LIN {X 0,Y 407.799,Z 694.938,A -85,B 0,C 180,E1 -11054.266,E2 -11054.266} C_VEL
LIN {X 0,Y 407.045,Z 706.099,A -85,B 0,C 180,E1 -11055.216,E2 -11055.216} C_VEL
LIN {X 0,Y 406.273,Z 716.85,A -85,B 0,C 180,E1 -11056.367,E2 -11056.367} C_VEL
LIN {X 0,Y 406.01,Z 720.118,A -85,B 0,C 180,E1 -11056.773,E2 -11056.773} C_VEL
LIN {X 0,Y 404.973,Z 724.447,A -85,B 0,C 180,E1 -11057.328,E2 -11057.328} C_VEL
LIN {X 0,Y 401.518,Z 731.114,A -85,B 0,C 180,E1 -11058.251,E2 -11058.251} C_VEL
LIN {X 0,Y 398.157,Z 737.243,A -85,B 0,C 180,E1 -11059.262,E2 -11059.262} C_VEL
LIN {X 0,Y 397.276,Z 740.61,A -85,B 0,C 180,E1 -11059.945,E2 -11059.945} C_VEL
LIN {X 0,Y 396.697,Z 746.419,A -85,B 0,C 180,E1 -11061.338,E2 -11061.338} C_VEL
LIN {X 0,Y 396.363,Z 751.512,A -85,B 0,C 180,E1 -11062.869,E2 -11062.869} C_VEL
LIN {X 0,Y 396.152,Z 755.462,A -85,B 0,C 180,E1 -11064.4,E2 -11064.4} C_VEL
LIN {X 0,Y 395.896,Z 758.382,A -85,B 0,C 180,E1 -11065.927,E2 -11065.927} C_VEL
LIN {X 0,Y 395.868,Z 759.782,A -85,B 0,C 180,E1 -11066.946,E2 -11066.946} C_VEL
LIN {X 0,Y 395.86,Z 760.777,A -85,B 0,C 180,E1 -11067.964,E2 -11067.964} C_VEL
LIN {X 0,Y 395.779,Z 761.627,A -85,B 0,C 180,E1 -11069.999,E2 -11069.999} C_VEL
LIN {X 0,Y 395.797,Z 761.439,A -85,B 0,C 180,E1 -11071.017,E2 -11071.017} C_VEL
LIN {X 0,Y 395.86,Z 760.855,A -85,B 0,C 180,E1 -11072.034,E2 -11072.034} C_VEL
LIN {X 0,Y 395.886,Z 758.539,A -85,B 0,C 180,E1 -11074.071,E2 -11074.071} C_VEL
LIN {X 0,Y 396.142,Z 755.67,A -85,B 0,C 180,E1 -11075.599,E2 -11075.599} C_VEL
LIN {X 0,Y 396.361,Z 751.784,A -85,B 0,C 180,E1 -11077.129,E2 -11077.129} C_VEL
LIN {X 0,Y 396.687,Z 746.775,A -85,B 0,C 180,E1 -11078.66,E2 -11078.66} C_VEL
LIN {X 0,Y 397.268,Z 740.464,A -85,B 0,C 180,E1 -11080.189,E2 -11080.189} C_VEL
LIN {X 0,Y 397.969,Z 732.562,A -85,B 0,C 180,E1 -11081.716,E2 -11081.716} C_VEL
LIN {X 0,Y 398.706,Z 724.506,A -85,B 0,C 180,E1 -11082.987,E2 -11082.987} C_VEL
LIN {X 0,Y 399.608,Z 714.671,A -85,B 0,C 180,E1 -11084.253,E2 -11084.253} C_VEL
LIN {X 0,Y 400.355,Z 703.619,A -85,B 0,C 180,E1 -11085.396,E2 -11085.396} C_VEL
LIN {X 0,Y 401.175,Z 692.77,A -85,B 0,C 180,E1 -11086.277,E2 -11086.277} C_VEL
LIN {X 0,Y 401.93,Z 680.778,A -85,B 0,C 180,E1 -11087.03,E2 -11087.03} C_VEL
LIN {X 0,Y 402.452,Z 668.5,A -85,B 0,C 180,E1 -11087.596,E2 -11087.596} C_VEL
LIN {X 0,Y 402.857,Z 655.856,A -85,B 0,C 180,E1 -11087.972,E2 -11087.972} C_VEL
LIN {X 0,Y 403.735,Z 572.554,A -85,B 0,C 180,E1 -11089.479,E2 -11089.479} C_VEL
LIN {X 0,Y 399.424,Z 551.598,A -85,B 0,C 180,E1 -11090.112,E2 -11090.112} C_VEL
LIN {X 0,Y 399.354,Z 550.806,A -85,B 0,C 180,E1 -11090.204,E2 -11090.204} C_VEL
LIN {X 0,Y 399.28,Z 546.202,A -85,B 0,C 180,E1 -11091.342,E2 -11091.342} C_VEL
LIN {X 0,Y 397.408,Z 536.356,A -85,B 0,C 180,E1 -11093.999,E2 -11093.999} C_VEL
LIN {X 0,Y 397.147,Z 535.042,A -85,B 0,C 180,E1 -11094.433,E2 -11094.433} C_VEL
LIN {X 0,Y 397.161,Z 535.013,A -85,B 0,C 180,E1 -11097.775,E2 -11097.775} C_VEL
LIN {X 0,Y 397.077,Z 535.02,A -85,B 0,C 180,E1 -11100.881,E2 -11100.881} C_VEL
LIN {X 0,Y 397.124,Z 535.017,A -85,B 0,C 180,E1 -11104.492,E2 -11104.492} C_VEL
LIN {X 0,Y 397.104,Z 535.018,A -85,B 0,C 180,E1 -11108.273,E2 -11108.273} C_VEL
LIN {X 0,Y 397.103,Z 535.014,A -85,B 0,C 180,E1 -11110.905,E2 -11110.905} C_VEL
LIN {X 0,Y 397.099,Z 535.014,A -85,B 0,C 180,E1 -11113.647,E2 -11113.647} C_VEL
LIN {X 0,Y 397.1,Z 535.015,A -85,B 0,C 180,E1 -11116.52,E2 -11116.52} C_VEL
LIN {X 0,Y 397.116,Z 535.011,A -85,B 0,C 180,E1 -11119.55,E2 -11119.55} C_VEL
LIN {X 0,Y 397.094,Z 535.008,A -85,B 0,C 180,E1 -11122.789,E2 -11122.789} C_VEL
LIN {X 0,Y 397.113,Z 535.015,A -85,B 0,C 180,E1 -11126.281,E2 -11126.281} C_VEL
LIN {X 0,Y 397.108,Z 535.017,A -85,B 0,C 180,E1 -11130.132,E2 -11130.132} C_VEL
LIN {X 0,Y 397.188,Z 534.999,A -85,B 0,C 180,E1 -11132.609,E2 -11132.609} C_VEL
LIN {X 0,Y 397.126,Z 535.013,A -85,B 0,C 180,E1 -11135.981,E2 -11135.981} C_VEL
LIN {X 0,Y 397.137,Z 535.017,A -85,B 0,C 180,E1 -11139.702,E2 -11139.702} C_VEL
LIN {X 0,Y 397.174,Z 535.005,A -85,B 0,C 180,E1 -11142.844,E2 -11142.844} C_VEL
LIN {X 0,Y 397.221,Z 535.002,A -85,B 0,C 180,E1 -11146.702,E2 -11146.702} C_VEL
LIN {X 0,Y 397.211,Z 534.997,A -85,B 0,C 180,E1 -11149.809,E2 -11149.809} C_VEL
LIN {X 0,Y 397.356,Z 534.985,A -85,B 0,C 180,E1 -11152.888,E2 -11152.888} C_VEL
LIN {X 0,Y 397.249,Z 534.999,A -85,B 0,C 180,E1 -11154.925,E2 -11154.925} C_VEL
LIN {X 0,Y 397.444,Z 534.974,A -85,B 0,C 180,E1 -11157.973,E2 -11157.973} C_VEL
LIN {X 0,Y 397.575,Z 534.96,A -85,B 0,C 180,E1 -11160,E2 -11160} C_VEL
LIN {X 0,Y 397.375,Z 534.979,A -85,B 0,C 180,E1 -11163.041,E2 -11163.041} C_VEL
LIN {X 0,Y 397.377,Z 534.984,A -85,B 0,C 180,E1 -11166.091,E2 -11166.091} C_VEL
LIN {X 0,Y 397.369,Z 534.982,A -85,B 0,C 180,E1 -11168.134,E2 -11168.134} C_VEL
LIN {X 0,Y 397.221,Z 535.002,A -85,B 0,C 180,E1 -11172.258,E2 -11172.258} C_VEL
LIN {X 0,Y 397.172,Z 535.007,A -85,B 0,C 180,E1 -11175.392,E2 -11175.392} C_VEL
LIN {X 0,Y 397.164,Z 535.009,A -85,B 0,C 180,E1 -11178.573,E2 -11178.573} C_VEL
LIN {X 0,Y 397.103,Z 535.015,A -85,B 0,C 180,E1 -11181.818,E2 -11181.818} C_VEL
LIN {X 0,Y 397.146,Z 535.015,A -85,B 0,C 180,E1 -11185.513,E2 -11185.513} C_VEL
LIN {X 0,Y 397.115,Z 535.016,A -85,B 0,C 180,E1 -11188.544,E2 -11188.544} C_VEL
LIN {X 0,Y 397.074,Z 535.023,A -85,B 0,C 180,E1 -11192.072,E2 -11192.072} C_VEL
LIN {X 0,Y 397.114,Z 535.008,A -85,B 0,C 180,E1 -11195.504,E2 -11195.504} C_VEL
LIN {X 0,Y 397.128,Z 535.013,A -85,B 0,C 180,E1 -11198.863,E2 -11198.863} C_VEL
LIN {X 0,Y 397.063,Z 535.012,A -85,B 0,C 180,E1 -11202.268,E2 -11202.268} C_VEL
LIN {X 0,Y 397.112,Z 535.018,A -85,B 0,C 180,E1 -11205.065,E2 -11205.065} C_VEL
LIN {X 0,Y 397.152,Z 535.013,A -85,B 0,C 180,E1 -11208.008,E2 -11208.008} C_VEL
LIN {X 0,Y 397.106,Z 534.998,A -85,B 0,C 180,E1 -11211.727,E2 -11211.727} C_VEL
LIN {X 0,Y 397.123,Z 535.016,A -85,B 0,C 180,E1 -11215.508,E2 -11215.508} C_VEL
LIN {X 0,Y 397.075,Z 534.966,A -85,B 0,C 180,E1 -11219.119,E2 -11219.119} C_VEL
LIN {X 0,Y 397.218,Z 535.203,A -85,B 0,C 180,E1 -11221.661,E2 -11221.661} C_VEL
LIN {X 0,Y 399.624,Z 546.906,A -85,B 0,C 180,E1 -11224.478,E2 -11224.478} C_VEL
LIN {X 0,Y 400.536,Z 552.863,A -85,B 0,C 180,E1 -11225.842,E2 -11225.842} C_VEL
LIN {X 0,Y 399.226,Z 569.505,A -85,B 0,C 180,E1 -11229.386,E2 -11229.386} C_VEL
LIN {X 0,Y 399.065,Z 572.109,A -85,B 0,C 180,E1 -11229.883,E2 -11229.883} C_VEL
LIN {X 0,Y 403.53,Z 599.626,A -85,B 0,C 180,E1 -11230.651,E2 -11230.651} C_VEL
LIN {X 0,Y 402.595,Z 680.184,A -85,B 0,C 180,E1 -11232.115,E2 -11232.115} C_VEL
LIN {X 0,Y 401.967,Z 693.403,A -85,B 0,C 180,E1 -11232.546,E2 -11232.546} C_VEL
LIN {X 0,Y 401.348,Z 705.547,A -85,B 0,C 180,E1 -11233.142,E2 -11233.142} C_VEL
LIN {X 0,Y 400.486,Z 717.81,A -85,B 0,C 180,E1 -11233.956,E2 -11233.956} C_VEL
LIN {X 0,Y 399.547,Z 729.658,A -85,B 0,C 180,E1 -11234.99,E2 -11234.99} C_VEL
LIN {X 0,Y 398.735,Z 739.944,A -85,B 0,C 180,E1 -11236.119,E2 -11236.119} C_VEL
LIN {X 0,Y 398.055,Z 748.375,A -85,B 0,C 180,E1 -11237.251,E2 -11237.251} C_VEL
LIN {X 0,Y 397.306,Z 756.249,A -85,B 0,C 180,E1 -11238.522,E2 -11238.522} C_VEL
LIN {X 0,Y 396.689,Z 763.945,A -85,B 0,C 180,E1 -11240.054,E2 -11240.054} C_VEL
LIN {X 0,Y 396.226,Z 771.041,A -85,B 0,C 180,E1 -11241.843,E2 -11241.843} C_VEL
LIN {X 0,Y 395.936,Z 775.764,A -85,B 0,C 180,E1 -11243.376,E2 -11243.376} C_VEL
LIN {X 0,Y 395.851,Z 779.377,A -85,B 0,C 180,E1 -11244.908,E2 -11244.908} C_VEL
LIN {X 0,Y 395.778,Z 781.239,A -85,B 0,C 180,E1 -11245.928,E2 -11245.928} C_VEL
LIN {X 0,Y 395.763,Z 783.631,A -85,B 0,C 180,E1 -11247.966,E2 -11247.966} C_VEL
LIN {X 0,Y 395.778,Z 784.939,A -85,B 0,C 180,E1 -11250.001,E2 -11250.001} C_VEL
LIN {X 0,Y 395.773,Z 784.842,A -85,B 0,C 180,E1 -11251.018,E2 -11251.018} C_VEL
LIN {X 0,Y 395.761,Z 784.158,A -85,B 0,C 180,E1 -11252.036,E2 -11252.036} C_VEL
LIN {X 0,Y 395.729,Z 782.89,A -85,B 0,C 180,E1 -11253.055,E2 -11253.055} C_VEL
LIN {X 0,Y 395.852,Z 779.359,A -85,B 0,C 180,E1 -11255.094,E2 -11255.094} C_VEL
LIN {X 0,Y 395.921,Z 775.744,A -85,B 0,C 180,E1 -11256.626,E2 -11256.626} C_VEL
LIN {X 0,Y 396.228,Z 771.015,A -85,B 0,C 180,E1 -11258.159,E2 -11258.159} C_VEL
LIN {X 0,Y 396.691,Z 763.91,A -85,B 0,C 180,E1 -11259.948,E2 -11259.948} C_VEL
LIN {X 0,Y 397.308,Z 756.204,A -85,B 0,C 180,E1 -11261.479,E2 -11261.479} C_VEL
LIN {X 0,Y 398.22,Z 746.53,A -85,B 0,C 180,E1 -11263.005,E2 -11263.005} C_VEL
LIN {X 0,Y 398.974,Z 736.549,A -85,B 0,C 180,E1 -11264.278,E2 -11264.278} C_VEL
LIN {X 0,Y 399.861,Z 725.275,A -85,B 0,C 180,E1 -11265.418,E2 -11265.418} C_VEL
LIN {X 0,Y 400.714,Z 714.238,A -85,B 0,C 180,E1 -11266.298,E2 -11266.298} C_VEL
LIN {X 0,Y 401.554,Z 702.011,A -85,B 0,C 180,E1 -11267.048,E2 -11267.048} C_VEL
LIN {X 0,Y 402.233,Z 689.149,A -85,B 0,C 180,E1 -11267.608,E2 -11267.608} C_VEL
LIN {X 0,Y 402.671,Z 675.476,A -85,B 0,C 180,E1 -11267.982,E2 -11267.982} C_VEL
LIN {X 0,Y 403.517,Z 599.547,A -85,B 0,C 180,E1 -11269.344,E2 -11269.344} C_VEL
LIN {X 0,Y 399.119,Z 572.48,A -85,B 0,C 180,E1 -11270.083,E2 -11270.083} C_VEL
LIN {X 0,Y 399.14,Z 570.706,A -85,B 0,C 180,E1 -11270.351,E2 -11270.351} C_VEL
LIN {X 0,Y 400.427,Z 554.441,A -85,B 0,C 180,E1 -11273.809,E2 -11273.809} C_VEL
LIN {X 0,Y 400.428,Z 551.46,A -85,B 0,C 180,E1 -11274.462,E2 -11274.462} C_VEL
LIN {X 0,Y 398.096,Z 539.235,A -85,B 0,C 180,E1 -11277.324,E2 -11277.324} C_VEL
LIN {X 0,Y 397.202,Z 535.088,A -85,B 0,C 180,E1 -11278.391,E2 -11278.391} C_VEL
LIN {X 0,Y 397.082,Z 535.023,A -85,B 0,C 180,E1 -11282.072,E2 -11282.072} C_VEL
LIN {X 0,Y 397.123,Z 535.016,A -85,B 0,C 180,E1 -11285.504,E2 -11285.504} C_VEL
LIN {X 0,Y 397.133,Z 535.013,A -85,B 0,C 180,E1 -11288.862,E2 -11288.862} C_VEL
LIN {X 0,Y 397.073,Z 535.023,A -85,B 0,C 180,E1 -11292.267,E2 -11292.267} C_VEL
LIN {X 0,Y 397.091,Z 535.022,A -85,B 0,C 180,E1 -11295.069,E2 -11295.069} C_VEL
LIN {X 0,Y 397.07,Z 535.024,A -85,B 0,C 180,E1 -11298.021,E2 -11298.021} C_VEL
LIN {X 0,Y 397.135,Z 535.015,A -85,B 0,C 180,E1 -11301.139,E2 -11301.139} C_VEL
LIN {X 0,Y 397.124,Z 535.018,A -85,B 0,C 180,E1 -11304.497,E2 -11304.497} C_VEL
LIN {X 0,Y 397.082,Z 535.025,A -85,B 0,C 180,E1 -11307.929,E2 -11307.929} C_VEL
LIN {X 0,Y 397.153,Z 535.328,A -85,B 0,C 180,E1 -11308.441,E2 -11308.441} C_VEL
LIN {X 0,Y 400.671,Z 546.972,A -85,B 0,C 180,E1 -11310.865,E2 -11310.865} C_VEL
LIN {X 0,Y 402.695,Z 556.853,A -85,B 0,C 180,E1 -11312.734,E2 -11312.734} C_VEL
LIN {X 0,Y 402.289,Z 566.911,A -85,B 0,C 180,E1 -11314.381,E2 -11314.381} C_VEL
LIN {X 0,Y 400.826,Z 591.579,A -85,B 0,C 180,E1 -11318.395,E2 -11318.395} C_VEL
LIN {X 0,Y 399.629,Z 613.667,A -85,B 0,C 180,E1 -11321.956,E2 -11321.956} C_VEL
LIN {X 0,Y 398.858,Z 631.986,A -85,B 0,C 180,E1 -11324.878,E2 -11324.878} C_VEL
LIN {X 0,Y 400.775,Z 645.77,A -85,B 0,C 180,E1 -11325.351,E2 -11325.351} C_VEL
LIN {X 0,Y 400.953,Z 651.079,A -85,B 0,C 180,E1 -11325.497,E2 -11325.497} C_VEL
LIN {X 0,Y 399.755,Z 704.823,A -85,B 0,C 180,E1 -11326.788,E2 -11326.788} C_VEL
LIN {X 0,Y 399.417,Z 714.365,A -85,B 0,C 180,E1 -11327.165,E2 -11327.165} C_VEL
LIN {X 0,Y 398.946,Z 725.525,A -85,B 0,C 180,E1 -11327.796,E2 -11327.796} C_VEL
LIN {X 0,Y 398.427,Z 735.11,A -85,B 0,C 180,E1 -11328.554,E2 -11328.554} C_VEL
LIN {X 0,Y 397.928,Z 743.939,A -85,B 0,C 180,E1 -11329.442,E2 -11329.442} C_VEL
LIN {X 0,Y 397.309,Z 752.78,A -85,B 0,C 180,E1 -11330.583,E2 -11330.583} C_VEL
LIN {X 0,Y 396.852,Z 759.018,A -85,B 0,C 180,E1 -11331.599,E2 -11331.599} C_VEL
LIN {X 0,Y 396.59,Z 764.139,A -85,B 0,C 180,E1 -11332.618,E2 -11332.618} C_VEL
LIN {X 0,Y 396.36,Z 769.29,A -85,B 0,C 180,E1 -11333.893,E2 -11333.893} C_VEL
LIN {X 0,Y 395.965,Z 773.837,A -85,B 0,C 180,E1 -11335.419,E2 -11335.419} C_VEL
LIN {X 0,Y 395.831,Z 776.856,A -85,B 0,C 180,E1 -11336.947,E2 -11336.947} C_VEL
LIN {X 0,Y 395.795,Z 778.116,A -85,B 0,C 180,E1 -11337.965,E2 -11337.965} C_VEL
LIN {X 0,Y 395.76,Z 778.793,A -85,B 0,C 180,E1 -11338.983,E2 -11338.983} C_VEL
LIN {X 0,Y 395.76,Z 778.896,A -85,B 0,C 180,E1 -11340,E2 -11340} C_VEL
LIN {X 0,Y 395.76,Z 778.422,A -85,B 0,C 180,E1 -11341.018,E2 -11341.018} C_VEL
LIN {X 0,Y 395.772,Z 777.361,A -85,B 0,C 180,E1 -11342.035,E2 -11342.035} C_VEL
LIN {X 0,Y 395.824,Z 774.538,A -85,B 0,C 180,E1 -11343.563,E2 -11343.563} C_VEL
LIN {X 0,Y 395.99,Z 770.335,A -85,B 0,C 180,E1 -11345.091,E2 -11345.091} C_VEL
LIN {X 0,Y 396.141,Z 764.731,A -85,B 0,C 180,E1 -11346.53,E2 -11346.53} C_VEL
LIN {X 0,Y 396.444,Z 759.18,A -85,B 0,C 180,E1 -11347.641,E2 -11347.641} C_VEL
LIN {X 0,Y 396.687,Z 752.914,A -85,B 0,C 180,E1 -11348.661,E2 -11348.661} C_VEL
LIN {X 0,Y 397.099,Z 744.072,A -85,B 0,C 180,E1 -11349.808,E2 -11349.808} C_VEL
LIN {X 0,Y 397.525,Z 735.203,A -85,B 0,C 180,E1 -11350.698,E2 -11350.698} C_VEL
LIN {X 0,Y 397.944,Z 725.554,A -85,B 0,C 180,E1 -11351.46,E2 -11351.46} C_VEL
LIN {X 0,Y 398.193,Z 715.643,A -85,B 0,C 180,E1 -11352.034,E2 -11352.034} C_VEL
LIN {X 0,Y 398.502,Z 705.429,A -85,B 0,C 180,E1 -11352.444,E2 -11352.444} C_VEL
LIN {X 0,Y 398.767,Z 689.785,A -85,B 0,C 180,E1 -11352.824,E2 -11352.824} C_VEL
LIN {X 0,Y 399.26,Z 646.715,A -85,B 0,C 180,E1 -11353.772,E2 -11353.772} C_VEL
LIN {X 0,Y 397.778,Z 631.757,A -85,B 0,C 180,E1 -11354.162,E2 -11354.162} C_VEL
LIN {X 0,Y 398.287,Z 617.682,A -85,B 0,C 180,E1 -11356.399,E2 -11356.399} C_VEL
LIN {X 0,Y 399.179,Z 596.662,A -85,B 0,C 180,E1 -11359.811,E2 -11359.811} C_VEL
LIN {X 0,Y 400.154,Z 575.39,A -85,B 0,C 180,E1 -11363.277,E2 -11363.277} C_VEL
LIN {X 0,Y 401.199,Z 556.319,A -85,B 0,C 180,E1 -11366.384,E2 -11366.384} C_VEL
LIN {X 0,Y 400.728,Z 551.948,A -85,B 0,C 180,E1 -11367.129,E2 -11367.129} C_VEL
LIN {X 0,Y 397.187,Z 535.186,A -85,B 0,C 180,E1 -11370.129,E2 -11370.129} C_VEL
LIN {X 0,Y 397.123,Z 535.018,A -85,B 0,C 180,E1 -11373.718,E2 -11373.718} C_VEL
LIN {X 0,Y 397.102,Z 535.018,A -85,B 0,C 180,E1 -11377.209,E2 -11377.209} C_VEL
LIN {X 0,Y 397.106,Z 535.008,A -85,B 0,C 180,E1 -11380.445,E2 -11380.445} C_VEL
LIN {X 0,Y 397.105,Z 534.994,A -85,B 0,C 180,E1 -11383.648,E2 -11383.648} C_VEL
LIN {X 0,Y 397.111,Z 535.02,A -85,B 0,C 180,E1 -11386.52,E2 -11386.52} C_VEL
LIN {X 0,Y 397.117,Z 534.998,A -85,B 0,C 180,E1 -11390.422,E2 -11390.422} C_VEL
LIN {X 0,Y 397.112,Z 535.02,A -85,B 0,C 180,E1 -11394.265,E2 -11394.265} C_VEL
LIN {X 0,Y 397.119,Z 535.017,A -85,B 0,C 180,E1 -11396.727,E2 -11396.727} C_VEL
LIN {X 0,Y 397.129,Z 535.019,A -85,B 0,C 180,E1 -11400.295,E2 -11400.295} C_VEL
LIN {X 0,Y 397.199,Z 535.011,A -85,B 0,C 180,E1 -11402.609,E2 -11402.609} C_VEL
LIN {X 0,Y 397.183,Z 535.091,A -85,B 0,C 180,E1 -11405.706,E2 -11405.706} C_VEL
LIN {X 0,Y 399.242,Z 545.825,A -85,B 0,C 180,E1 -11408.659,E2 -11408.659} C_VEL
LIN {X 0,Y 399.384,Z 550.325,A -85,B 0,C 180,E1 -11409.797,E2 -11409.797} C_VEL
LIN {X 0,Y 399.383,Z 551.427,A -85,B 0,C 180,E1 -11409.978,E2 -11409.978} C_VEL
LIN {X 0,Y 403.8,Z 572.909,A -85,B 0,C 180,E1 -11410.629,E2 -11410.629} C_VEL
LIN {X 0,Y 402.826,Z 655.828,A -85,B 0,C 180,E1 -11412.123,E2 -11412.123} C_VEL
LIN {X 0,Y 402.425,Z 668.491,A -85,B 0,C 180,E1 -11412.499,E2 -11412.499} C_VEL
LIN {X 0,Y 401.831,Z 681.338,A -85,B 0,C 180,E1 -11413.095,E2 -11413.095} C_VEL
LIN {X 0,Y 401.117,Z 693.197,A -85,B 0,C 180,E1 -11413.85,E2 -11413.85} C_VEL
LIN {X 0,Y 400.352,Z 703.959,A -85,B 0,C 180,E1 -11414.732,E2 -11414.732} C_VEL
LIN {X 0,Y 399.589,Z 714.927,A -85,B 0,C 180,E1 -11415.874,E2 -11415.874} C_VEL
LIN {X 0,Y 398.584,Z 725.605,A -85,B 0,C 180,E1 -11417.266,E2 -11417.266} C_VEL
LIN {X 0,Y 397.941,Z 733.475,A -85,B 0,C 180,E1 -11418.539,E2 -11418.539} C_VEL
LIN {X 0,Y 397.276,Z 740.61,A -85,B 0,C 180,E1 -11419.945,E2 -11419.945} C_VEL
LIN {X 0,Y 396.419,Z 743.788,A -85,B 0,C 180,E1 -11420.653,E2 -11420.653} C_VEL
LIN {X 0,Y 393.189,Z 748.517,A -85,B 0,C 180,E1 -11421.826,E2 -11421.826} C_VEL
LIN {X 0,Y 389.965,Z 752.575,A -85,B 0,C 180,E1 -11423.067,E2 -11423.067} C_VEL
LIN {X 0,Y 389.14,Z 754.668,A -85,B 0,C 180,E1 -11423.873,E2 -11423.873} C_VEL
LIN {X 0,Y 388.822,Z 758.588,A -85,B 0,C 180,E1 -11425.853,E2 -11425.853} C_VEL
LIN {X 0,Y 388.772,Z 759.987,A -85,B 0,C 180,E1 -11426.89,E2 -11426.89} C_VEL
LIN {X 0,Y 388.763,Z 760.982,A -85,B 0,C 180,E1 -11427.927,E2 -11427.927} C_VEL
LIN {X 0,Y 388.708,Z 761.831,A -85,B 0,C 180,E1 -11429.999,E2 -11429.999} C_VEL
LIN {X 0,Y 388.728,Z 761.643,A -85,B 0,C 180,E1 -11431.035,E2 -11431.035} C_VEL
LIN {X 0,Y 388.762,Z 761.06,A -85,B 0,C 180,E1 -11432.071,E2 -11432.071} C_VEL
LIN {X 0,Y 388.812,Z 758.743,A -85,B 0,C 180,E1 -11434.145,E2 -11434.145} C_VEL
LIN {X 0,Y 389.075,Z 755.874,A -85,B 0,C 180,E1 -11435.701,E2 -11435.701} C_VEL
LIN {X 0,Y 389.312,Z 751.987,A -85,B 0,C 180,E1 -11437.259,E2 -11437.259} C_VEL
LIN {X 0,Y 389.672,Z 746.978,A -85,B 0,C 180,E1 -11438.817,E2 -11438.817} C_VEL
LIN {X 0,Y 390.281,Z 740.667,A -85,B 0,C 180,E1 -11440.373,E2 -11440.373} C_VEL
LIN {X 0,Y 391.009,Z 732.764,A -85,B 0,C 180,E1 -11441.928,E2 -11441.928} C_VEL
LIN {X 0,Y 391.804,Z 724.707,A -85,B 0,C 180,E1 -11443.22,E2 -11443.22} C_VEL
LIN {X 0,Y 392.723,Z 714.872,A -85,B 0,C 180,E1 -11444.508,E2 -11444.508} C_VEL
LIN {X 0,Y 393.51,Z 703.818,A -85,B 0,C 180,E1 -11445.671,E2 -11445.671} C_VEL
LIN {X 0,Y 394.387,Z 692.968,A -85,B 0,C 180,E1 -11446.565,E2 -11446.565} C_VEL
LIN {X 0,Y 395.159,Z 680.975,A -85,B 0,C 180,E1 -11447.331,E2 -11447.331} C_VEL
LIN {X 0,Y 395.712,Z 668.692,A -85,B 0,C 180,E1 -11447.906,E2 -11447.906} C_VEL
LIN {X 0,Y 396.129,Z 656.038,A -85,B 0,C 180,E1 -11448.288,E2 -11448.288} C_VEL
LIN {X 0,Y 397.126,Z 573.966,A -85,B 0,C 180,E1 -11449.793,E2 -11449.793} C_VEL
LIN {X 0,Y 392.54,Z 551.801,A -85,B 0,C 180,E1 -11450.48,E2 -11450.48} C_VEL
LIN {X 0,Y 392.484,Z 551.002,A -85,B 0,C 180,E1 -11450.573,E2 -11450.573} C_VEL
LIN {X 0,Y 392.23,Z 546.783,A -85,B 0,C 180,E1 -11451.647,E2 -11451.647} C_VEL
LIN {X 0,Y 390.217,Z 536.551,A -85,B 0,C 180,E1 -11454.47,E2 -11454.47} C_VEL
LIN {X 0,Y 390.124,Z 535.905,A -85,B 0,C 180,E1 -11454.76,E2 -11454.76} C_VEL
LIN {X 0,Y 390.095,Z 535.892,A -85,B 0,C 180,E1 -11458.019,E2 -11458.019} C_VEL
LIN {X 0,Y 390.022,Z 535.905,A -85,B 0,C 180,E1 -11461.503,E2 -11461.503} C_VEL
LIN {X 0,Y 390.066,Z 535.898,A -85,B 0,C 180,E1 -11464.024,E2 -11464.024} C_VEL
LIN {X 0,Y 390.043,Z 535.903,A -85,B 0,C 180,E1 -11467.55,E2 -11467.55} C_VEL
LIN {X 0,Y 390.068,Z 535.89,A -85,B 0,C 180,E1 -11470.823,E2 -11470.823} C_VEL
LIN {X 0,Y 390.053,Z 535.889,A -85,B 0,C 180,E1 -11473.885,E2 -11473.885} C_VEL
LIN {X 0,Y 390.076,Z 535.898,A -85,B 0,C 180,E1 -11477.619,E2 -11477.619} C_VEL
LIN {X 0,Y 390.09,Z 535.878,A -85,B 0,C 180,E1 -11480.907,E2 -11480.907} C_VEL
LIN {X 0,Y 390.081,Z 535.892,A -85,B 0,C 180,E1 -11484.792,E2 -11484.792} C_VEL
LIN {X 0,Y 390.021,Z 535.897,A -85,B 0,C 180,E1 -11488.495,E2 -11488.495} C_VEL
LIN {X 0,Y 390.11,Z 535.882,A -85,B 0,C 180,E1 -11492.069,E2 -11492.069} C_VEL
LIN {X 0,Y 390.074,Z 535.897,A -85,B 0,C 180,E1 -11495.519,E2 -11495.519} C_VEL
LIN {X 0,Y 390.054,Z 535.89,A -85,B 0,C 180,E1 -11498.878,E2 -11498.878} C_VEL
LIN {X 0,Y 390.121,Z 535.883,A -85,B 0,C 180,E1 -11502.166,E2 -11502.166} C_VEL
LIN {X 0,Y 390.136,Z 535.883,A -85,B 0,C 180,E1 -11505.392,E2 -11505.392} C_VEL
LIN {X 0,Y 390.141,Z 535.881,A -85,B 0,C 180,E1 -11508.571,E2 -11508.571} C_VEL
LIN {X 0,Y 390.336,Z 535.861,A -85,B 0,C 180,E1 -11511.993,E2 -11511.993} C_VEL
LIN {X 0,Y 390.221,Z 535.874,A -85,B 0,C 180,E1 -11514.833,E2 -11514.833} C_VEL
LIN {X 0,Y 390.413,Z 535.85,A -85,B 0,C 180,E1 -11517.937,E2 -11517.937} C_VEL
LIN {X 0,Y 390.544,Z 535.836,A -85,B 0,C 180,E1 -11520,E2 -11520} C_VEL
LIN {X 0,Y 390.309,Z 535.86,A -85,B 0,C 180,E1 -11523.097,E2 -11523.097} C_VEL
LIN {X 0,Y 390.33,Z 535.861,A -85,B 0,C 180,E1 -11526.202,E2 -11526.202} C_VEL
LIN {X 0,Y 390.307,Z 535.861,A -85,B 0,C 180,E1 -11528.282,E2 -11528.282} C_VEL
LIN {X 0,Y 390.17,Z 535.88,A -85,B 0,C 180,E1 -11532.483,E2 -11532.483} C_VEL
LIN {X 0,Y 390.132,Z 535.881,A -85,B 0,C 180,E1 -11535.677,E2 -11535.677} C_VEL
LIN {X 0,Y 390.109,Z 535.889,A -85,B 0,C 180,E1 -11538.922,E2 -11538.922} C_VEL
LIN {X 0,Y 390.041,Z 535.894,A -85,B 0,C 180,E1 -11542.234,E2 -11542.234} C_VEL
LIN {X 0,Y 390.112,Z 535.887,A -85,B 0,C 180,E1 -11545.744,E2 -11545.744} C_VEL
LIN {X 0,Y 390.052,Z 535.898,A -85,B 0,C 180,E1 -11549.11,E2 -11549.11} C_VEL
LIN {X 0,Y 390.037,Z 535.898,A -85,B 0,C 180,E1 -11552.722,E2 -11552.722} C_VEL
LIN {X 0,Y 390.051,Z 535.883,A -85,B 0,C 180,E1 -11555.826,E2 -11555.826} C_VEL
LIN {X 0,Y 390.066,Z 535.895,A -85,B 0,C 180,E1 -11559.22,E2 -11559.22} C_VEL
LIN {X 0,Y 390.037,Z 535.887,A -85,B 0,C 180,E1 -11562.375,E2 -11562.375} C_VEL
LIN {X 0,Y 390.097,Z 535.887,A -85,B 0,C 180,E1 -11566.108,E2 -11566.108} C_VEL
LIN {X 0,Y 390.079,Z 535.895,A -85,B 0,C 180,E1 -11569.175,E2 -11569.175} C_VEL
LIN {X 0,Y 390.044,Z 535.876,A -85,B 0,C 180,E1 -11572.449,E2 -11572.449} C_VEL
LIN {X 0,Y 390.065,Z 535.888,A -85,B 0,C 180,E1 -11575.976,E2 -11575.976} C_VEL
LIN {X 0,Y 390.035,Z 535.847,A -85,B 0,C 180,E1 -11579.701,E2 -11579.701} C_VEL
LIN {X 0,Y 390.136,Z 536.007,A -85,B 0,C 180,E1 -11581.309,E2 -11581.309} C_VEL
LIN {X 0,Y 392.112,Z 545.401,A -85,B 0,C 180,E1 -11583.66,E2 -11583.66} C_VEL
LIN {X 0,Y 393.588,Z 553.612,A -85,B 0,C 180,E1 -11585.598,E2 -11585.598} C_VEL
LIN {X 0,Y 392.572,Z 566.29,A -85,B 0,C 180,E1 -11588.356,E2 -11588.356} C_VEL
LIN {X 0,Y 392.171,Z 571.907,A -85,B 0,C 180,E1 -11589.513,E2 -11589.513} C_VEL
LIN {X 0,Y 396.631,Z 598.893,A -85,B 0,C 180,E1 -11590.29,E2 -11590.29} C_VEL
LIN {X 0,Y 396.898,Z 604.479,A -85,B 0,C 180,E1 -11590.409,E2 -11590.409} C_VEL
LIN {X 0,Y 395.847,Z 679.991,A -85,B 0,C 180,E1 -11591.799,E2 -11591.799} C_VEL
LIN {X 0,Y 395.19,Z 693.206,A -85,B 0,C 180,E1 -11592.237,E2 -11592.237} C_VEL
LIN {X 0,Y 394.542,Z 705.348,A -85,B 0,C 180,E1 -11592.842,E2 -11592.842} C_VEL
LIN {X 0,Y 393.66,Z 717.61,A -85,B 0,C 180,E1 -11593.67,E2 -11593.67} C_VEL
LIN {X 0,Y 392.709,Z 729.2,A -85,B 0,C 180,E1 -11594.696,E2 -11594.696} C_VEL
LIN {X 0,Y 391.826,Z 739.797,A -85,B 0,C 180,E1 -11595.876,E2 -11595.876} C_VEL
LIN {X 0,Y 391.118,Z 748.172,A -85,B 0,C 180,E1 -11597.021,E2 -11597.021} C_VEL
LIN {X 0,Y 390.316,Z 756.045,A -85,B 0,C 180,E1 -11598.314,E2 -11598.314} C_VEL
LIN {X 0,Y 389.672,Z 763.741,A -85,B 0,C 180,E1 -11599.873,E2 -11599.873} C_VEL
LIN {X 0,Y 389.158,Z 770.836,A -85,B 0,C 180,E1 -11601.694,E2 -11601.694} C_VEL
LIN {X 0,Y 388.852,Z 775.558,A -85,B 0,C 180,E1 -11603.254,E2 -11603.254} C_VEL
LIN {X 0,Y 388.746,Z 779.172,A -85,B 0,C 180,E1 -11604.815,E2 -11604.815} C_VEL
LIN {X 0,Y 388.703,Z 781.035,A -85,B 0,C 180,E1 -11605.854,E2 -11605.854} C_VEL
LIN {X 0,Y 388.661,Z 783.428,A -85,B 0,C 180,E1 -11607.928,E2 -11607.928} C_VEL
LIN {X 0,Y 388.703,Z 784.331,A -85,B 0,C 180,E1 -11608.965,E2 -11608.965} C_VEL
LIN {X 0,Y 388.707,Z 784.857,A -85,B 0,C 180,E1 -11610.001,E2 -11610.001} C_VEL
LIN {X 0,Y 388.672,Z 784.808,A -85,B 0,C 180,E1 -11611.037,E2 -11611.037} C_VEL
LIN {X 0,Y 388.658,Z 784.172,A -85,B 0,C 180,E1 -11612.073,E2 -11612.073} C_VEL
LIN {X 0,Y 388.636,Z 782.944,A -85,B 0,C 180,E1 -11613.111,E2 -11613.111} C_VEL
LIN {X 0,Y 388.733,Z 777.962,A -85,B 0,C 180,E1 -11615.762,E2 -11615.762} C_VEL
LIN {X 0,Y 388.942,Z 774.103,A -85,B 0,C 180,E1 -11617.267,E2 -11617.267} C_VEL
LIN {X 0,Y 389.357,Z 767.984,A -85,B 0,C 180,E1 -11619.088,E2 -11619.088} C_VEL
LIN {X 0,Y 389.881,Z 761.302,A -85,B 0,C 180,E1 -11620.648,E2 -11620.648} C_VEL
LIN {X 0,Y 390.633,Z 753.015,A -85,B 0,C 180,E1 -11622.205,E2 -11622.205} C_VEL
LIN {X 0,Y 391.403,Z 744.52,A -85,B 0,C 180,E1 -11623.5,E2 -11623.5} C_VEL
LIN {X 0,Y 392.242,Z 734.022,A -85,B 0,C 180,E1 -11624.794,E2 -11624.794} C_VEL
LIN {X 0,Y 393.136,Z 723.638,A -85,B 0,C 180,E1 -11625.821,E2 -11625.821} C_VEL
LIN {X 0,Y 394.061,Z 712.261,A -85,B 0,C 180,E1 -11626.714,E2 -11626.714} C_VEL
LIN {X 0,Y 394.828,Z 700.579,A -85,B 0,C 180,E1 -11627.414,E2 -11627.414} C_VEL
LIN {X 0,Y 395.562,Z 687.102,A -85,B 0,C 180,E1 -11627.982,E2 -11627.982} C_VEL
LIN {X 0,Y 395.981,Z 673.712,A -85,B 0,C 180,E1 -11628.33,E2 -11628.33} C_VEL
LIN {X 0,Y 396.796,Z 600.305,A -85,B 0,C 180,E1 -11629.666,E2 -11629.666} C_VEL
LIN {X 0,Y 392.212,Z 571.997,A -85,B 0,C 180,E1 -11630.469,E2 -11630.469} C_VEL
LIN {X 0,Y 392.46,Z 567.476,A -85,B 0,C 180,E1 -11631.378,E2 -11631.378} C_VEL
LIN {X 0,Y 393.635,Z 554.251,A -85,B 0,C 180,E1 -11634.246,E2 -11634.246} C_VEL
LIN {X 0,Y 392.105,Z 545.375,A -85,B 0,C 180,E1 -11636.338,E2 -11636.338} C_VEL
LIN {X 0,Y 390.189,Z 536.144,A -85,B 0,C 180,E1 -11638.621,E2 -11638.621} C_VEL
LIN {X 0,Y 390.092,Z 535.868,A -85,B 0,C 180,E1 -11639.108,E2 -11639.108} C_VEL
LIN {X 0,Y 390.047,Z 535.901,A -85,B 0,C 180,E1 -11642.722,E2 -11642.722} C_VEL
LIN {X 0,Y 390.06,Z 535.897,A -85,B 0,C 180,E1 -11645.826,E2 -11645.826} C_VEL
LIN {X 0,Y 390.073,Z 535.893,A -85,B 0,C 180,E1 -11649.219,E2 -11649.219} C_VEL
LIN {X 0,Y 390.046,Z 535.898,A -85,B 0,C 180,E1 -11652.375,E2 -11652.375} C_VEL
LIN {X 0,Y 390.048,Z 535.9,A -85,B 0,C 180,E1 -11655.355,E2 -11655.355} C_VEL
LIN {X 0,Y 390.035,Z 535.901,A -85,B 0,C 180,E1 -11658.187,E2 -11658.187} C_VEL
LIN {X 0,Y 390.095,Z 535.892,A -85,B 0,C 180,E1 -11660.908,E2 -11660.908} C_VEL
LIN {X 0,Y 390.09,Z 535.894,A -85,B 0,C 180,E1 -11664.794,E2 -11664.794} C_VEL
LIN {X 0,Y 390.071,Z 536.13,A -85,B 0,C 180,E1 -11667.712,E2 -11667.712} C_VEL
LIN {X 0,Y 393.337,Z 546.37,A -85,B 0,C 180,E1 -11669.98,E2 -11669.98} C_VEL
LIN {X 0,Y 395.349,Z 554.413,A -85,B 0,C 180,E1 -11671.607,E2 -11671.607} C_VEL
LIN {X 0,Y 396.227,Z 560.862,A -85,B 0,C 180,E1 -11672.804,E2 -11672.804} C_VEL
LIN {X 0,Y 394.864,Z 580.85,A -85,B 0,C 180,E1 -11676.114,E2 -11676.114} C_VEL
LIN {X 0,Y 393.769,Z 598.994,A -85,B 0,C 180,E1 -11679.086,E2 -11679.086} C_VEL
LIN {X 0,Y 392.542,Z 621.651,A -85,B 0,C 180,E1 -11682.818,E2 -11682.818} C_VEL
LIN {X 0,Y 392.053,Z 631.777,A -85,B 0,C 180,E1 -11684.46,E2 -11684.46} C_VEL
LIN {X 0,Y 393.839,Z 644.005,A -85,B 0,C 180,E1 -11684.923,E2 -11684.923} C_VEL
LIN {X 0,Y 394.362,Z 650.095,A -85,B 0,C 180,E1 -11685.113,E2 -11685.113} C_VEL
LIN {X 0,Y 393.043,Z 704.735,A -85,B 0,C 180,E1 -11686.46,E2 -11686.46} C_VEL
LIN {X 0,Y 392.628,Z 714.914,A -85,B 0,C 180,E1 -11686.873,E2 -11686.873} C_VEL
LIN {X 0,Y 392.203,Z 724.906,A -85,B 0,C 180,E1 -11687.451,E2 -11687.451} C_VEL
LIN {X 0,Y 391.621,Z 734.613,A -85,B 0,C 180,E1 -11688.221,E2 -11688.221} C_VEL
LIN {X 0,Y 391.171,Z 742.32,A -85,B 0,C 180,E1 -11688.995,E2 -11688.995} C_VEL
LIN {X 0,Y 390.591,Z 749.696,A -85,B 0,C 180,E1 -11689.896,E2 -11689.896} C_VEL
LIN {X 0,Y 389.968,Z 758.074,A -85,B 0,C 180,E1 -11691.188,E2 -11691.188} C_VEL
LIN {X 0,Y 389.65,Z 763.372,A -85,B 0,C 180,E1 -11692.225,E2 -11692.225} C_VEL
LIN {X 0,Y 389.327,Z 768.622,A -85,B 0,C 180,E1 -11693.504,E2 -11693.504} C_VEL
LIN {X 0,Y 389.032,Z 772.798,A -85,B 0,C 180,E1 -11694.818,E2 -11694.818} C_VEL
LIN {X 0,Y 388.817,Z 775.246,A -85,B 0,C 180,E1 -11695.854,E2 -11695.854} C_VEL
LIN {X 0,Y 388.737,Z 777.05,A -85,B 0,C 180,E1 -11696.891,E2 -11696.891} C_VEL
LIN {X 0,Y 388.698,Z 778.254,A -85,B 0,C 180,E1 -11697.928,E2 -11697.928} C_VEL
LIN {X 0,Y 388.66,Z 778.878,A -85,B 0,C 180,E1 -11698.964,E2 -11698.964} C_VEL
LIN {X 0,Y 388.672,Z 778.928,A -85,B 0,C 180,E1 -11700,E2 -11700} C_VEL
LIN {X 0,Y 388.66,Z 778.401,A -85,B 0,C 180,E1 -11701.036,E2 -11701.036} C_VEL
LIN {X 0,Y 388.671,Z 777.293,A -85,B 0,C 180,E1 -11702.073,E2 -11702.073} C_VEL
LIN {X 0,Y 388.738,Z 774.403,A -85,B 0,C 180,E1 -11703.628,E2 -11703.628} C_VEL
LIN {X 0,Y 388.868,Z 771.681,A -85,B 0,C 180,E1 -11704.665,E2 -11704.665} C_VEL
LIN {X 0,Y 388.942,Z 768.227,A -85,B 0,C 180,E1 -11705.704,E2 -11705.704} C_VEL
LIN {X 0,Y 389.197,Z 762.779,A -85,B 0,C 180,E1 -11707.001,E2 -11707.001} C_VEL
LIN {X 0,Y 389.481,Z 755.731,A -85,B 0,C 180,E1 -11708.3,E2 -11708.3} C_VEL
LIN {X 0,Y 389.824,Z 748.577,A -85,B 0,C 180,E1 -11709.338,E2 -11709.338} C_VEL
LIN {X 0,Y 390.285,Z 739.727,A -85,B 0,C 180,E1 -11710.374,E2 -11710.374} C_VEL
LIN {X 0,Y 390.738,Z 729.517,A -85,B 0,C 180,E1 -11711.28,E2 -11711.28} C_VEL
LIN {X 0,Y 391.083,Z 719.927,A -85,B 0,C 180,E1 -11711.927,E2 -11711.927} C_VEL
LIN {X 0,Y 391.409,Z 708.481,A -85,B 0,C 180,E1 -11712.476,E2 -11712.476} C_VEL
LIN {X 0,Y 391.566,Z 697.509,A -85,B 0,C 180,E1 -11712.8,E2 -11712.8} C_VEL
LIN {X 0,Y 392.325,Z 647.718,A -85,B 0,C 180,E1 -11713.916,E2 -11713.916} C_VEL
LIN {X 0,Y 390.787,Z 631.502,A -85,B 0,C 180,E1 -11714.367,E2 -11714.367} C_VEL
LIN {X 0,Y 391.636,Z 609.264,A -85,B 0,C 180,E1 -11717.991,E2 -11717.991} C_VEL
LIN {X 0,Y 392.618,Z 588.297,A -85,B 0,C 180,E1 -11721.436,E2 -11721.436} C_VEL
LIN {X 0,Y 393.777,Z 566.331,A -85,B 0,C 180,E1 -11725.052,E2 -11725.052} C_VEL
LIN {X 0,Y 394.237,Z 556.093,A -85,B 0,C 180,E1 -11726.752,E2 -11726.752} C_VEL
LIN {X 0,Y 391.388,Z 541.814,A -85,B 0,C 180,E1 -11729.296,E2 -11729.296} C_VEL
LIN {X 0,Y 390.122,Z 536.021,A -85,B 0,C 180,E1 -11730.386,E2 -11730.386} C_VEL
LIN {X 0,Y 390.073,Z 535.898,A -85,B 0,C 180,E1 -11734.024,E2 -11734.024} C_VEL
LIN {X 0,Y 390.05,Z 535.897,A -85,B 0,C 180,E1 -11737.551,E2 -11737.551} C_VEL
LIN {X 0,Y 390.06,Z 535.88,A -85,B 0,C 180,E1 -11740.821,E2 -11740.821} C_VEL
LIN {X 0,Y 390.059,Z 535.872,A -85,B 0,C 180,E1 -11743.886,E2 -11743.886} C_VEL
LIN {X 0,Y 390.068,Z 535.894,A -85,B 0,C 180,E1 -11747.622,E2 -11747.622} C_VEL
LIN {X 0,Y 390.093,Z 535.873,A -85,B 0,C 180,E1 -11750.907,E2 -11750.907} C_VEL
LIN {X 0,Y 390.089,Z 535.887,A -85,B 0,C 180,E1 -11754.793,E2 -11754.793} C_VEL
LIN {X 0,Y 390.028,Z 535.898,A -85,B 0,C 180,E1 -11758.495,E2 -11758.495} C_VEL
LIN {X 0,Y 390.122,Z 535.889,A -85,B 0,C 180,E1 -11762.07,E2 -11762.07} C_VEL
LIN {X 0,Y 390.144,Z 536.012,A -85,B 0,C 180,E1 -11765.452,E2 -11765.452} C_VEL
LIN {X 0,Y 392.36,Z 547.553,A -85,B 0,C 180,E1 -11768.66,E2 -11768.66} C_VEL
LIN {X 0,Y 392.488,Z 551.37,A -85,B 0,C 180,E1 -11769.587,E2 -11769.587} C_VEL
LIN {X 0,Y 394.157,Z 559.358,A -85,B 0,C 180,E1 -11769.872,E2 -11769.872} C_VEL
LIN {X 0,Y 397.182,Z 575.064,A -85,B 0,C 180,E1 -11770.329,E2 -11770.329} C_VEL
LIN {X 0,Y 396.001,Z 657.527,A -85,B 0,C 180,E1 -11771.838,E2 -11771.838} C_VEL
LIN {X 0,Y 395.575,Z 671.012,A -85,B 0,C 180,E1 -11772.286,E2 -11772.286} C_VEL
LIN {X 0,Y 394.895,Z 683.806,A -85,B 0,C 180,E1 -11772.922,E2 -11772.922} C_VEL
LIN {X 0,Y 394.191,Z 695.149,A -85,B 0,C 180,E1 -11773.691,E2 -11773.691} C_VEL
LIN {X 0,Y 393.35,Z 706.065,A -85,B 0,C 180,E1 -11774.642,E2 -11774.642} C_VEL
LIN {X 0,Y 392.511,Z 717.267,A -85,B 0,C 180,E1 -11775.879,E2 -11775.879} C_VEL
LIN {X 0,Y 391.661,Z 725.813,A -85,B 0,C 180,E1 -11777.037,E2 -11777.037} C_VEL
LIN {X 0,Y 390.987,Z 733.682,A -85,B 0,C 180,E1 -11778.332,E2 -11778.332} C_VEL
LIN {X 0,Y 390.25,Z 741.374,A -85,B 0,C 180,E1 -11779.886,E2 -11779.886} C_VEL
LIN {X 0,Y 389.497,Z 748.436,A -85,B 0,C 180,E1 -11781.699,E2 -11781.699} C_VEL
LIN {X 0,Y 389.193,Z 753.27,A -85,B 0,C 180,E1 -11783.308,E2 -11783.308} C_VEL
LIN {X 0,Y 389.14,Z 754.668,A -85,B 0,C 180,E1 -11783.873,E2 -11783.873} C_VEL
LIN {X 0,Y 388.357,Z 756.529,A -85,B 0,C 180,E1 -11784.692,E2 -11784.692} C_VEL
LIN {X 0,Y 385.332,Z 759.013,A -85,B 0,C 180,E1 -11786.041,E2 -11786.041} C_VEL
LIN {X 0,Y 382.819,Z 760.483,A -85,B 0,C 180,E1 -11787.148,E2 -11787.148} C_VEL
LIN {X 0,Y 381.735,Z 761.281,A -85,B 0,C 180,E1 -11788.016,E2 -11788.016} C_VEL
LIN {X 0,Y 381.642,Z 761.433,A -85,B 0,C 180,E1 -11788.311,E2 -11788.311} C_VEL
LIN {X 0,Y 381.64,Z 762.035,A -85,B 0,C 180,E1 -11789.999,E2 -11789.999} C_VEL
LIN {X 0,Y 381.644,Z 761.847,A -85,B 0,C 180,E1 -11791.054,E2 -11791.054} C_VEL
LIN {X 0,Y 381.665,Z 761.264,A -85,B 0,C 180,E1 -11792.11,E2 -11792.11} C_VEL
LIN {X 0,Y 381.743,Z 758.946,A -85,B 0,C 180,E1 -11794.222,E2 -11794.222} C_VEL
LIN {X 0,Y 382.01,Z 756.077,A -85,B 0,C 180,E1 -11795.806,E2 -11795.806} C_VEL
LIN {X 0,Y 382.257,Z 752.191,A -85,B 0,C 180,E1 -11797.393,E2 -11797.393} C_VEL
LIN {X 0,Y 382.646,Z 747.181,A -85,B 0,C 180,E1 -11798.981,E2 -11798.981} C_VEL
LIN {X 0,Y 383.286,Z 740.869,A -85,B 0,C 180,E1 -11800.565,E2 -11800.565} C_VEL
LIN {X 0,Y 384.05,Z 732.966,A -85,B 0,C 180,E1 -11802.147,E2 -11802.147} C_VEL
LIN {X 0,Y 384.895,Z 724.909,A -85,B 0,C 180,E1 -11803.461,E2 -11803.461} C_VEL
LIN {X 0,Y 385.851,Z 715.073,A -85,B 0,C 180,E1 -11804.772,E2 -11804.772} C_VEL
LIN {X 0,Y 386.672,Z 704.018,A -85,B 0,C 180,E1 -11805.955,E2 -11805.955} C_VEL
LIN {X 0,Y 387.598,Z 693.166,A -85,B 0,C 180,E1 -11806.864,E2 -11806.864} C_VEL
LIN {X 0,Y 388.398,Z 681.171,A -85,B 0,C 180,E1 -11807.642,E2 -11807.642} C_VEL
LIN {X 0,Y 388.947,Z 667.997,A -85,B 0,C 180,E1 -11808.262,E2 -11808.262} C_VEL
LIN {X 0,Y 389.436,Z 654.718,A -85,B 0,C 180,E1 -11808.647,E2 -11808.647} C_VEL
LIN {X 0,Y 390.499,Z 575.18,A -85,B 0,C 180,E1 -11810.123,E2 -11810.123} C_VEL
LIN {X 0,Y 385.68,Z 552.124,A -85,B 0,C 180,E1 -11810.854,E2 -11810.854} C_VEL
LIN {X 0,Y 385.576,Z 551.2,A -85,B 0,C 180,E1 -11810.959,E2 -11810.959} C_VEL
LIN {X 0,Y 384.938,Z 546.297,A -85,B 0,C 180,E1 -11812.261,E2 -11812.261} C_VEL
LIN {X 0,Y 383.103,Z 536.819,A -85,B 0,C 180,E1 -11814.992,E2 -11814.992} C_VEL
LIN {X 0,Y 383.016,Z 536.767,A -85,B 0,C 180,E1 -11818.493,E2 -11818.493} C_VEL
LIN {X 0,Y 383.007,Z 536.774,A -85,B 0,C 180,E1 -11822.148,E2 -11822.148} C_VEL
LIN {X 0,Y 383.016,Z 536.775,A -85,B 0,C 180,E1 -11824.667,E2 -11824.667} C_VEL
LIN {X 0,Y 382.999,Z 536.777,A -85,B 0,C 180,E1 -11827.903,E2 -11827.903} C_VEL
LIN {X 0,Y 382.994,Z 536.776,A -85,B 0,C 180,E1 -11831.344,E2 -11831.344} C_VEL
LIN {X 0,Y 382.994,Z 536.766,A -85,B 0,C 180,E1 -11834.303,E2 -11834.303} C_VEL
LIN {X 0,Y 383.035,Z 536.771,A -85,B 0,C 180,E1 -11837.243,E2 -11837.243} C_VEL
LIN {X 0,Y 383.017,Z 536.761,A -85,B 0,C 180,E1 -11840.411,E2 -11840.411} C_VEL
LIN {X 0,Y 383.022,Z 536.772,A -85,B 0,C 180,E1 -11844.044,E2 -11844.044} C_VEL
LIN {X 0,Y 383.006,Z 536.772,A -85,B 0,C 180,E1 -11846.599,E2 -11846.599} C_VEL
LIN {X 0,Y 382.992,Z 536.775,A -85,B 0,C 180,E1 -11850.3,E2 -11850.3} C_VEL
LIN {X 0,Y 383.05,Z 536.76,A -85,B 0,C 180,E1 -11852.697,E2 -11852.697} C_VEL
LIN {X 0,Y 383.027,Z 536.768,A -85,B 0,C 180,E1 -11856.192,E2 -11856.192} C_VEL
LIN {X 0,Y 383.053,Z 536.77,A -85,B 0,C 180,E1 -11859.598,E2 -11859.598} C_VEL
LIN {X 0,Y 383.097,Z 536.758,A -85,B 0,C 180,E1 -11862.931,E2 -11862.931} C_VEL
LIN {X 0,Y 383.117,Z 536.758,A -85,B 0,C 180,E1 -11866.463,E2 -11866.463} C_VEL
LIN {X 0,Y 383.144,Z 536.746,A -85,B 0,C 180,E1 -11870.498,E2 -11870.498} C_VEL
LIN {X 0,Y 383.265,Z 536.74,A -85,B 0,C 180,E1 -11872.625,E2 -11872.625} C_VEL
LIN {X 0,Y 383.193,Z 536.749,A -85,B 0,C 180,E1 -11874.738,E2 -11874.738} C_VEL
LIN {X 0,Y 383.38,Z 536.725,A -85,B 0,C 180,E1 -11877.899,E2 -11877.899} C_VEL
LIN {X 0,Y 383.514,Z 536.712,A -85,B 0,C 180,E1 -11880,E2 -11880} C_VEL
LIN {X 0,Y 383.245,Z 536.739,A -85,B 0,C 180,E1 -11883.154,E2 -11883.154} C_VEL
LIN {X 0,Y 383.286,Z 536.738,A -85,B 0,C 180,E1 -11886.316,E2 -11886.316} C_VEL
LIN {X 0,Y 383.252,Z 536.739,A -85,B 0,C 180,E1 -11888.436,E2 -11888.436} C_VEL
LIN {X 0,Y 383.1,Z 536.761,A -85,B 0,C 180,E1 -11891.642,E2 -11891.642} C_VEL
LIN {X 0,Y 383.104,Z 536.759,A -85,B 0,C 180,E1 -11894.882,E2 -11894.882} C_VEL
LIN {X 0,Y 383.086,Z 536.764,A -85,B 0,C 180,E1 -11898.172,E2 -11898.172} C_VEL
LIN {X 0,Y 382.997,Z 536.772,A -85,B 0,C 180,E1 -11901.531,E2 -11901.531} C_VEL
LIN {X 0,Y 383.045,Z 536.769,A -85,B 0,C 180,E1 -11904.961,E2 -11904.961} C_VEL
LIN {X 0,Y 383.023,Z 536.773,A -85,B 0,C 180,E1 -11908.271,E2 -11908.271} C_VEL
LIN {X 0,Y 383.005,Z 536.775,A -85,B 0,C 180,E1 -11912.15,E2 -11912.15} C_VEL
LIN {X 0,Y 383.012,Z 536.769,A -85,B 0,C 180,E1 -11914.669,E2 -11914.669} C_VEL
LIN {X 0,Y 382.996,Z 536.769,A -85,B 0,C 180,E1 -11917.905,E2 -11917.905} C_VEL
LIN {X 0,Y 382.979,Z 536.775,A -85,B 0,C 180,E1 -11921.348,E2 -11921.348} C_VEL
LIN {X 0,Y 383.003,Z 536.776,A -85,B 0,C 180,E1 -11924.306,E2 -11924.306} C_VEL
LIN {X 0,Y 383.071,Z 536.76,A -85,B 0,C 180,E1 -11927.25,E2 -11927.25} C_VEL
LIN {X 0,Y 383.019,Z 536.766,A -85,B 0,C 180,E1 -11930.413,E2 -11930.413} C_VEL
LIN {X 0,Y 383.024,Z 536.77,A -85,B 0,C 180,E1 -11934.046,E2 -11934.046} C_VEL
LIN {X 0,Y 382.983,Z 536.729,A -85,B 0,C 180,E1 -11937.579,E2 -11937.579} C_VEL
LIN {X 0,Y 383.09,Z 536.898,A -85,B 0,C 180,E1 -11940.988,E2 -11940.988} C_VEL
LIN {X 0,Y 385.234,Z 547.113,A -85,B 0,C 180,E1 -11943.592,E2 -11943.592} C_VEL
LIN {X 0,Y 386.672,Z 555.157,A -85,B 0,C 180,E1 -11945.529,E2 -11945.529} C_VEL
LIN {X 0,Y 385.451,Z 569.101,A -85,B 0,C 180,E1 -11948.614,E2 -11948.614} C_VEL
LIN {X 0,Y 385.321,Z 571.743,A -85,B 0,C 180,E1 -11949.136,E2 -11949.136} C_VEL
LIN {X 0,Y 389.888,Z 599.245,A -85,B 0,C 180,E1 -11949.945,E2 -11949.945} C_VEL
LIN {X 0,Y 390.212,Z 604.293,A -85,B 0,C 180,E1 -11950.059,E2 -11950.059} C_VEL
LIN {X 0,Y 389.119,Z 679.799,A -85,B 0,C 180,E1 -11951.473,E2 -11951.473} C_VEL
LIN {X 0,Y 388.449,Z 693.01,A -85,B 0,C 180,E1 -11951.918,E2 -11951.918} C_VEL
LIN {X 0,Y 387.74,Z 705.149,A -85,B 0,C 180,E1 -11952.531,E2 -11952.531} C_VEL
LIN {X 0,Y 386.857,Z 717.409,A -85,B 0,C 180,E1 -11953.375,E2 -11953.375} C_VEL
LIN {X 0,Y 385.845,Z 728.996,A -85,B 0,C 180,E1 -11954.416,E2 -11954.416} C_VEL
LIN {X 0,Y 384.972,Z 738.936,A -85,B 0,C 180,E1 -11955.536,E2 -11955.536} C_VEL
LIN {X 0,Y 384.174,Z 747.969,A -85,B 0,C 180,E1 -11956.782,E2 -11956.782} C_VEL
LIN {X 0,Y 383.347,Z 755.842,A -85,B 0,C 180,E1 -11958.098,E2 -11958.098} C_VEL
LIN {X 0,Y 382.668,Z 763.537,A -85,B 0,C 180,E1 -11959.686,E2 -11959.686} C_VEL
LIN {X 0,Y 382.107,Z 770.632,A -85,B 0,C 180,E1 -11961.54,E2 -11961.54} C_VEL
LIN {X 0,Y 381.785,Z 775.354,A -85,B 0,C 180,E1 -11963.129,E2 -11963.129} C_VEL
LIN {X 0,Y 381.647,Z 778.968,A -85,B 0,C 180,E1 -11964.718,E2 -11964.718} C_VEL
LIN {X 0,Y 381.628,Z 780.831,A -85,B 0,C 180,E1 -11965.777,E2 -11965.777} C_VEL
LIN {X 0,Y 381.56,Z 783.226,A -85,B 0,C 180,E1 -11967.89,E2 -11967.89} C_VEL
LIN {X 0,Y 381.62,Z 784.767,A -85,B 0,C 180,E1 -11970.001,E2 -11970.001} C_VEL
LIN {X 0,Y 381.571,Z 784.781,A -85,B 0,C 180,E1 -11971.056,E2 -11971.056} C_VEL
LIN {X 0,Y 381.556,Z 784.204,A -85,B 0,C 180,E1 -11972.112,E2 -11972.112} C_VEL
LIN {X 0,Y 381.548,Z 783.032,A -85,B 0,C 180,E1 -11973.169,E2 -11973.169} C_VEL
LIN {X 0,Y 381.629,Z 780.067,A -85,B 0,C 180,E1 -11974.755,E2 -11974.755} C_VEL
LIN {X 0,Y 381.782,Z 775.33,A -85,B 0,C 180,E1 -11976.873,E2 -11976.873} C_VEL
LIN {X 0,Y 382.109,Z 770.601,A -85,B 0,C 180,E1 -11978.462,E2 -11978.462} C_VEL
LIN {X 0,Y 382.67,Z 763.496,A -85,B 0,C 180,E1 -11980.316,E2 -11980.316} C_VEL
LIN {X 0,Y 383.349,Z 755.789,A -85,B 0,C 180,E1 -11981.903,E2 -11981.903} C_VEL
LIN {X 0,Y 384.315,Z 746.114,A -85,B 0,C 180,E1 -11983.484,E2 -11983.484} C_VEL
LIN {X 0,Y 385.171,Z 736.132,A -85,B 0,C 180,E1 -11984.801,E2 -11984.801} C_VEL
LIN {X 0,Y 386.174,Z 724.858,A -85,B 0,C 180,E1 -11985.978,E2 -11985.978} C_VEL
LIN {X 0,Y 387.123,Z 713.82,A -85,B 0,C 180,E1 -11986.887,E2 -11986.887} C_VEL
LIN {X 0,Y 387.999,Z 701.589,A -85,B 0,C 180,E1 -11987.663,E2 -11987.663} C_VEL
LIN {X 0,Y 388.719,Z 688.719,A -85,B 0,C 180,E1 -11988.241,E2 -11988.241} C_VEL
LIN {X 0,Y 389.188,Z 675.034,A -85,B 0,C 180,E1 -11988.628,E2 -11988.628} C_VEL
LIN {X 0,Y 390.12,Z 601.181,A -85,B 0,C 180,E1 -11989.996,E2 -11989.996} C_VEL
LIN {X 0,Y 385.354,Z 572.026,A -85,B 0,C 180,E1 -11990.835,E2 -11990.835} C_VEL
LIN {X 0,Y 385.332,Z 570.971,A -85,B 0,C 180,E1 -11990.975,E2 -11990.975} C_VEL
LIN {X 0,Y 386.601,Z 556.57,A -85,B 0,C 180,E1 -11994.141,E2 -11994.141} C_VEL
LIN {X 0,Y 386.331,Z 552.787,A -85,B 0,C 180,E1 -11995.022,E2 -11995.022} C_VEL
LIN {X 0,Y 384.122,Z 541.381,A -85,B 0,C 180,E1 -11997.812,E2 -11997.812} C_VEL
LIN {X 0,Y 383.08,Z 536.867,A -85,B 0,C 180,E1 -11999.015,E2 -11999.015} C_VEL
LIN {X 0,Y 382.991,Z 536.779,A -85,B 0,C 180,E1 -12002.423,E2 -12002.423} C_VEL
LIN {X 0,Y 383.029,Z 536.774,A -85,B 0,C 180,E1 -12005.956,E2 -12005.956} C_VEL
LIN {X 0,Y 383.019,Z 536.774,A -85,B 0,C 180,E1 -12009.587,E2 -12009.587} C_VEL
LIN {X 0,Y 383.009,Z 536.774,A -85,B 0,C 180,E1 -12012.779,E2 -12012.779} C_VEL
LIN {X 0,Y 383.001,Z 536.777,A -85,B 0,C 180,E1 -12015.79,E2 -12015.79} C_VEL
LIN {X 0,Y 382.992,Z 536.779,A -85,B 0,C 180,E1 -12018.796,E2 -12018.796} C_VEL
LIN {X 0,Y 383.005,Z 536.777,A -85,B 0,C 180,E1 -12022.096,E2 -12022.096} C_VEL
LIN {X 0,Y 383.022,Z 536.776,A -85,B 0,C 180,E1 -12025.332,E2 -12025.332} C_VEL
LIN {X 0,Y 383.052,Z 537.027,A -85,B 0,C 180,E1 -12026.94,E2 -12026.94} C_VEL
LIN {X 0,Y 386.514,Z 547.534,A -85,B 0,C 180,E1 -12029.394,E2 -12029.394} C_VEL
LIN {X 0,Y 388.918,Z 557.062,A -85,B 0,C 180,E1 -12031.388,E2 -12031.388} C_VEL
LIN {X 0,Y 389.724,Z 562.548,A -85,B 0,C 180,E1 -12032.452,E2 -12032.452} C_VEL
LIN {X 0,Y 388.335,Z 581.764,A -85,B 0,C 180,E1 -12035.687,E2 -12035.687} C_VEL
LIN {X 0,Y 387.033,Z 601.465,A -85,B 0,C 180,E1 -12038.984,E2 -12038.984} C_VEL
LIN {X 0,Y 385.712,Z 624.17,A -85,B 0,C 180,E1 -12042.777,E2 -12042.777} C_VEL
LIN {X 0,Y 385.309,Z 631.788,A -85,B 0,C 180,E1 -12044.02,E2 -12044.02} C_VEL
LIN {X 0,Y 387.25,Z 644.336,A -85,B 0,C 180,E1 -12044.525,E2 -12044.525} C_VEL
LIN {X 0,Y 387.772,Z 650.613,A -85,B 0,C 180,E1 -12044.733,E2 -12044.733} C_VEL
LIN {X 0,Y 386.284,Z 705.556,A -85,B 0,C 180,E1 -12046.151,E2 -12046.151} C_VEL
LIN {X 0,Y 385.875,Z 715.497,A -85,B 0,C 180,E1 -12046.572,E2 -12046.572} C_VEL
LIN {X 0,Y 385.359,Z 726.221,A -85,B 0,C 180,E1 -12047.225,E2 -12047.225} C_VEL
LIN {X 0,Y 384.728,Z 735.652,A -85,B 0,C 180,E1 -12048.007,E2 -12048.007} C_VEL
LIN {X 0,Y 384.178,Z 744.379,A -85,B 0,C 180,E1 -12048.926,E2 -12048.926} C_VEL
LIN {X 0,Y 383.553,Z 752.28,A -85,B 0,C 180,E1 -12049.975,E2 -12049.975} C_VEL
LIN {X 0,Y 382.986,Z 758.613,A -85,B 0,C 180,E1 -12051.026,E2 -12051.026} C_VEL
LIN {X 0,Y 382.556,Z 764.98,A -85,B 0,C 180,E1 -12052.346,E2 -12052.346} C_VEL
LIN {X 0,Y 382.27,Z 769.987,A -85,B 0,C 180,E1 -12053.667,E2 -12053.667} C_VEL
LIN {X 0,Y 381.989,Z 773.096,A -85,B 0,C 180,E1 -12054.722,E2 -12054.722} C_VEL
LIN {X 0,Y 381.748,Z 775.499,A -85,B 0,C 180,E1 -12055.777,E2 -12055.777} C_VEL
LIN {X 0,Y 381.645,Z 777.252,A -85,B 0,C 180,E1 -12056.833,E2 -12056.833} C_VEL
LIN {X 0,Y 381.6,Z 778.401,A -85,B 0,C 180,E1 -12057.889,E2 -12057.889} C_VEL
LIN {X 0,Y 381.561,Z 778.967,A -85,B 0,C 180,E1 -12058.945,E2 -12058.945} C_VEL
LIN {X 0,Y 381.573,Z 778.956,A -85,B 0,C 180,E1 -12060,E2 -12060} C_VEL
LIN {X 0,Y 381.559,Z 778.366,A -85,B 0,C 180,E1 -12061.055,E2 -12061.055} C_VEL
LIN {X 0,Y 381.57,Z 777.188,A -85,B 0,C 180,E1 -12062.111,E2 -12062.111} C_VEL
LIN {X 0,Y 381.657,Z 774.226,A -85,B 0,C 180,E1 -12063.695,E2 -12063.695} C_VEL
LIN {X 0,Y 381.814,Z 769.818,A -85,B 0,C 180,E1 -12065.281,E2 -12065.281} C_VEL
LIN {X 0,Y 381.93,Z 765.408,A -85,B 0,C 180,E1 -12066.446,E2 -12066.446} C_VEL
LIN {X 0,Y 382.237,Z 759.625,A -85,B 0,C 180,E1 -12067.661,E2 -12067.661} C_VEL
LIN {X 0,Y 382.523,Z 753.417,A -85,B 0,C 180,E1 -12068.718,E2 -12068.718} C_VEL
LIN {X 0,Y 382.93,Z 744.719,A -85,B 0,C 180,E1 -12069.908,E2 -12069.908} C_VEL
LIN {X 0,Y 383.383,Z 735.961,A -85,B 0,C 180,E1 -12070.83,E2 -12070.83} C_VEL
LIN {X 0,Y 383.796,Z 726.473,A -85,B 0,C 180,E1 -12071.621,E2 -12071.621} C_VEL
LIN {X 0,Y 384.126,Z 715.724,A -85,B 0,C 180,E1 -12072.28,E2 -12072.28} C_VEL
LIN {X 0,Y 384.453,Z 705.636,A -85,B 0,C 180,E1 -12072.705,E2 -12072.705} C_VEL
LIN {X 0,Y 384.757,Z 687.622,A -85,B 0,C 180,E1 -12073.165,E2 -12073.165} C_VEL
LIN {X 0,Y 385.291,Z 647.982,A -85,B 0,C 180,E1 -12074.086,E2 -12074.086} C_VEL
LIN {X 0,Y 383.729,Z 631.708,A -85,B 0,C 180,E1 -12074.528,E2 -12074.528} C_VEL
LIN {X 0,Y 384.592,Z 611.645,A -85,B 0,C 180,E1 -12077.824,E2 -12077.824} C_VEL
LIN {X 0,Y 385.582,Z 590.241,A -85,B 0,C 180,E1 -12081.379,E2 -12081.379} C_VEL
LIN {X 0,Y 386.853,Z 566.866,A -85,B 0,C 180,E1 -12085.273,E2 -12085.273} C_VEL
LIN {X 0,Y 387.325,Z 558.402,A -85,B 0,C 180,E1 -12086.685,E2 -12086.685} C_VEL
LIN {X 0,Y 386.171,Z 551.349,A -85,B 0,C 180,E1 -12087.945,E2 -12087.945} C_VEL
LIN {X 0,Y 383.087,Z 536.891,A -85,B 0,C 180,E1 -12090.617,E2 -12090.617} C_VEL
LIN {X 0,Y 383.023,Z 536.776,A -85,B 0,C 180,E1 -12094.668,E2 -12094.668} C_VEL
LIN {X 0,Y 383.006,Z 536.775,A -85,B 0,C 180,E1 -12097.904,E2 -12097.904} C_VEL
LIN {X 0,Y 382.988,Z 536.757,A -85,B 0,C 180,E1 -12101.347,E2 -12101.347} C_VEL
LIN {X 0,Y 383.001,Z 536.754,A -85,B 0,C 180,E1 -12104.303,E2 -12104.303} C_VEL
LIN {X 0,Y 383.014,Z 536.773,A -85,B 0,C 180,E1 -12107.24,E2 -12107.24} C_VEL
LIN {X 0,Y 383.019,Z 536.752,A -85,B 0,C 180,E1 -12110.413,E2 -12110.413} C_VEL
LIN {X 0,Y 383.029,Z 536.773,A -85,B 0,C 180,E1 -12114.044,E2 -12114.044} C_VEL
LIN {X 0,Y 382.991,Z 536.777,A -85,B 0,C 180,E1 -12117.577,E2 -12117.577} C_VEL
LIN {X 0,Y 382.997,Z 536.78,A -85,B 0,C 180,E1 -12120.3,E2 -12120.3} C_VEL
LIN {X 0,Y 383.085,Z 536.767,A -85,B 0,C 180,E1 -12124.02,E2 -12124.02} C_VEL
LIN {X 0,Y 383.115,Z 536.954,A -85,B 0,C 180,E1 -12125.188,E2 -12125.188} C_VEL
LIN {X 0,Y 385.362,Z 548.515,A -85,B 0,C 180,E1 -12128.452,E2 -12128.452} C_VEL
LIN {X 0,Y 385.616,Z 551.583,A -85,B 0,C 180,E1 -12129.207,E2 -12129.207} C_VEL
LIN {X 0,Y 387.37,Z 559.66,A -85,B 0,C 180,E1 -12129.504,E2 -12129.504} C_VEL
LIN {X 0,Y 390.509,Z 575.473,A -85,B 0,C 180,E1 -12129.983,E2 -12129.983} C_VEL
LIN {X 0,Y 389.273,Z 657.751,A -85,B 0,C 180,E1 -12131.513,E2 -12131.513} C_VEL
LIN {X 0,Y 388.836,Z 671.227,A -85,B 0,C 180,E1 -12131.969,E2 -12131.969} C_VEL
LIN {X 0,Y 388.138,Z 684.018,A -85,B 0,C 180,E1 -12132.616,E2 -12132.616} C_VEL
LIN {X 0,Y 387.4,Z 695.36,A -85,B 0,C 180,E1 -12133.397,E2 -12133.397} C_VEL
LIN {X 0,Y 386.481,Z 706.626,A -85,B 0,C 180,E1 -12134.4,E2 -12134.4} C_VEL
LIN {X 0,Y 385.644,Z 717.475,A -85,B 0,C 180,E1 -12135.622,E2 -12135.622} C_VEL
LIN {X 0,Y 384.754,Z 726.021,A -85,B 0,C 180,E1 -12136.801,E2 -12136.801} C_VEL
LIN {X 0,Y 384.024,Z 733.89,A -85,B 0,C 180,E1 -12138.118,E2 -12138.118} C_VEL
LIN {X 0,Y 383.245,Z 741.581,A -85,B 0,C 180,E1 -12139.699,E2 -12139.699} C_VEL
LIN {X 0,Y 382.477,Z 748.643,A -85,B 0,C 180,E1 -12141.546,E2 -12141.546} C_VEL
LIN {X 0,Y 382.109,Z 753.834,A -85,B 0,C 180,E1 -12143.318,E2 -12143.318} C_VEL
LIN {X 0,Y 381.954,Z 756.933,A -85,B 0,C 180,E1 -12144.72,E2 -12144.72} C_VEL
LIN {X 0,Y 381.751,Z 758.793,A -85,B 0,C 180,E1 -12145.776,E2 -12145.776} C_VEL
LIN {X 0,Y 381.678,Z 760.193,A -85,B 0,C 180,E1 -12146.832,E2 -12146.832} C_VEL
LIN {X 0,Y 381.642,Z 761.433,A -85,B 0,C 180,E1 -12148.311,E2 -12148.311} C_VEL
LIN {X 0,Y 380.951,Z 761.927,A -85,B 0,C 180,E1 -12149.19,E2 -12149.19} C_VEL
LIN {X 0,Y 378.064,Z 762.061,A -85,B 0,C 180,E1 -12150.621,E2 -12150.621} C_VEL
LIN {X 0,Y 375.647,Z 761.701,A -85,B 0,C 180,E1 -12151.778,E2 -12151.778} C_VEL
LIN {X 0,Y 374.58,Z 760.926,A -85,B 0,C 180,E1 -12152.818,E2 -12152.818} C_VEL
LIN {X 0,Y 374.566,Z 760.735,A -85,B 0,C 180,E1 -12152.969,E2 -12152.969} C_VEL
LIN {X 0,Y 374.677,Z 759.15,A -85,B 0,C 180,E1 -12154.302,E2 -12154.302} C_VEL
LIN {X 0,Y 374.947,Z 756.281,A -85,B 0,C 180,E1 -12155.916,E2 -12155.916} C_VEL
LIN {X 0,Y 375.194,Z 752.395,A -85,B 0,C 180,E1 -12157.533,E2 -12157.533} C_VEL
LIN {X 0,Y 375.638,Z 747.384,A -85,B 0,C 180,E1 -12159.15,E2 -12159.15} C_VEL
LIN {X 0,Y 376.299,Z 741.072,A -85,B 0,C 180,E1 -12160.763,E2 -12160.763} C_VEL
LIN {X 0,Y 377.108,Z 733.169,A -85,B 0,C 180,E1 -12162.375,E2 -12162.375} C_VEL
LIN {X 0,Y 377.984,Z 725.11,A -85,B 0,C 180,E1 -12163.712,E2 -12163.712} C_VEL
LIN {X 0,Y 379.007,Z 715.273,A -85,B 0,C 180,E1 -12165.045,E2 -12165.045} C_VEL
LIN {X 0,Y 379.846,Z 704.218,A -85,B 0,C 180,E1 -12166.25,E2 -12166.25} C_VEL
LIN {X 0,Y 380.822,Z 693.364,A -85,B 0,C 180,E1 -12167.173,E2 -12167.173} C_VEL
LIN {X 0,Y 381.644,Z 681.367,A -85,B 0,C 180,E1 -12167.965,E2 -12167.965} C_VEL
LIN {X 0,Y 382.216,Z 669.077,A -85,B 0,C 180,E1 -12168.561,E2 -12168.561} C_VEL
LIN {X 0,Y 382.724,Z 656.403,A -85,B 0,C 180,E1 -12168.952,E2 -12168.952} C_VEL
LIN {X 0,Y 383.848,Z 576.307,A -85,B 0,C 180,E1 -12170.469,E2 -12170.469} C_VEL
LIN {X 0,Y 379.101,Z 553.666,A -85,B 0,C 180,E1 -12171.19,E2 -12171.19} C_VEL
LIN {X 0,Y 378.641,Z 551.504,A -85,B 0,C 180,E1 -12171.338,E2 -12171.338} C_VEL
LIN {X 0,Y 376.906,Z 542.032,A -85,B 0,C 180,E1 -12173.98,E2 -12173.98} C_VEL
LIN {X 0,Y 376.053,Z 537.685,A -85,B 0,C 180,E1 -12175.308,E2 -12175.308} C_VEL
LIN {X 0,Y 375.959,Z 537.64,A -85,B 0,C 180,E1 -12179.079,E2 -12179.079} C_VEL
LIN {X 0,Y 375.949,Z 537.652,A -85,B 0,C 180,E1 -12182.827,E2 -12182.827} C_VEL
LIN {X 0,Y 375.956,Z 537.651,A -85,B 0,C 180,E1 -12185.414,E2 -12185.414} C_VEL
LIN {X 0,Y 375.973,Z 537.65,A -85,B 0,C 180,E1 -12188.27,E2 -12188.27} C_VEL
LIN {X 0,Y 375.941,Z 537.658,A -85,B 0,C 180,E1 -12191.602,E2 -12191.602} C_VEL
LIN {X 0,Y 375.924,Z 537.645,A -85,B 0,C 180,E1 -12195.267,E2 -12195.267} C_VEL
LIN {X 0,Y 375.956,Z 537.652,A -85,B 0,C 180,E1 -12198.394,E2 -12198.394} C_VEL
LIN {X 0,Y 375.973,Z 537.634,A -85,B 0,C 180,E1 -12201.728,E2 -12201.728} C_VEL
LIN {X 0,Y 375.983,Z 537.653,A -85,B 0,C 180,E1 -12205.33,E2 -12205.33} C_VEL
LIN {X 0,Y 375.954,Z 537.649,A -85,B 0,C 180,E1 -12208.437,E2 -12208.437} C_VEL
LIN {X 0,Y 375.996,Z 537.639,A -85,B 0,C 180,E1 -12212.141,E2 -12212.141} C_VEL
LIN {X 0,Y 375.999,Z 537.646,A -85,B 0,C 180,E1 -12214.538,E2 -12214.538} C_VEL
LIN {X 0,Y 375.958,Z 537.646,A -85,B 0,C 180,E1 -12218.045,E2 -12218.045} C_VEL
LIN {X 0,Y 376.017,Z 537.647,A -85,B 0,C 180,E1 -12221.473,E2 -12221.473} C_VEL
LIN {X 0,Y 376.051,Z 537.633,A -85,B 0,C 180,E1 -12224.832,E2 -12224.832} C_VEL
LIN {X 0,Y 376.042,Z 537.638,A -85,B 0,C 180,E1 -12228.136,E2 -12228.136} C_VEL
LIN {X 0,Y 376.25,Z 537.617,A -85,B 0,C 180,E1 -12231.877,E2 -12231.877} C_VEL
LIN {X 0,Y 376.165,Z 537.624,A -85,B 0,C 180,E1 -12234.64,E2 -12234.64} C_VEL
LIN {X 0,Y 376.346,Z 537.6,A -85,B 0,C 180,E1 -12237.86,E2 -12237.86} C_VEL
LIN {X 0,Y 376.483,Z 537.588,A -85,B 0,C 180,E1 -12240,E2 -12240} C_VEL
LIN {X 0,Y 376.183,Z 537.617,A -85,B 0,C 180,E1 -12243.213,E2 -12243.213} C_VEL
LIN {X 0,Y 376.244,Z 537.615,A -85,B 0,C 180,E1 -12246.435,E2 -12246.435} C_VEL
LIN {X 0,Y 376.198,Z 537.618,A -85,B 0,C 180,E1 -12248.595,E2 -12248.595} C_VEL
LIN {X 0,Y 376.051,Z 537.642,A -85,B 0,C 180,E1 -12251.863,E2 -12251.863} C_VEL
LIN {X 0,Y 376.052,Z 537.639,A -85,B 0,C 180,E1 -12255.168,E2 -12255.168} C_VEL
LIN {X 0,Y 376.022,Z 537.643,A -85,B 0,C 180,E1 -12258.526,E2 -12258.526} C_VEL
LIN {X 0,Y 375.964,Z 537.648,A -85,B 0,C 180,E1 -12261.954,E2 -12261.954} C_VEL
LIN {X 0,Y 376,Z 537.649,A -85,B 0,C 180,E1 -12265.462,E2 -12265.462} C_VEL
LIN {X 0,Y 375.954,Z 537.654,A -85,B 0,C 180,E1 -12269.081,E2 -12269.081} C_VEL
LIN {X 0,Y 375.945,Z 537.653,A -85,B 0,C 180,E1 -12272.829,E2 -12272.829} C_VEL
LIN {X 0,Y 375.952,Z 537.643,A -85,B 0,C 180,E1 -12275.416,E2 -12275.416} C_VEL
LIN {X 0,Y 375.971,Z 537.65,A -85,B 0,C 180,E1 -12278.272,E2 -12278.272} C_VEL
LIN {X 0,Y 375.929,Z 537.649,A -85,B 0,C 180,E1 -12281.602,E2 -12281.602} C_VEL
LIN {X 0,Y 375.974,Z 537.653,A -85,B 0,C 180,E1 -12285.262,E2 -12285.262} C_VEL
LIN {X 0,Y 375.985,Z 537.65,A -85,B 0,C 180,E1 -12288.391,E2 -12288.391} C_VEL
LIN {X 0,Y 375.964,Z 537.628,A -85,B 0,C 180,E1 -12291.913,E2 -12291.913} C_VEL
LIN {X 0,Y 375.977,Z 537.652,A -85,B 0,C 180,E1 -12295.334,E2 -12295.334} C_VEL
LIN {X 0,Y 375.937,Z 537.595,A -85,B 0,C 180,E1 -12298.437,E2 -12298.437} C_VEL
LIN {X 0,Y 376.005,Z 537.725,A -85,B 0,C 180,E1 -12300.618,E2 -12300.618} C_VEL
LIN {X 0,Y 376.971,Z 541.934,A -85,B 0,C 180,E1 -12301.784,E2 -12301.784} C_VEL
LIN {X 0,Y 379.358,Z 553.905,A -85,B 0,C 180,E1 -12304.781,E2 -12304.781} C_VEL
LIN {X 0,Y 379.709,Z 557.121,A -85,B 0,C 180,E1 -12305.553,E2 -12305.553} C_VEL
LIN {X 0,Y 378.437,Z 571.324,A -85,B 0,C 180,E1 -12308.716,E2 -12308.716} C_VEL
LIN {X 0,Y 379.392,Z 577.089,A -85,B 0,C 180,E1 -12308.932,E2 -12308.932} C_VEL
LIN {X 0,Y 383.525,Z 602.38,A -85,B 0,C 180,E1 -12309.663,E2 -12309.663} C_VEL
LIN {X 0,Y 382.406,Z 679.607,A -85,B 0,C 180,E1 -12311.136,E2 -12311.136} C_VEL
LIN {X 0,Y 381.718,Z 692.814,A -85,B 0,C 180,E1 -12311.588,E2 -12311.588} C_VEL
LIN {X 0,Y 380.978,Z 704.95,A -85,B 0,C 180,E1 -12312.211,E2 -12312.211} C_VEL
LIN {X 0,Y 380.055,Z 717.209,A -85,B 0,C 180,E1 -12313.068,E2 -12313.068} C_VEL
LIN {X 0,Y 378.988,Z 728.794,A -85,B 0,C 180,E1 -12314.127,E2 -12314.127} C_VEL
LIN {X 0,Y 377.994,Z 739.584,A -85,B 0,C 180,E1 -12315.372,E2 -12315.372} C_VEL
LIN {X 0,Y 377.236,Z 747.766,A -85,B 0,C 180,E1 -12316.535,E2 -12316.535} C_VEL
LIN {X 0,Y 376.391,Z 755.638,A -85,B 0,C 180,E1 -12317.875,E2 -12317.875} C_VEL
LIN {X 0,Y 375.657,Z 763.333,A -85,B 0,C 180,E1 -12319.491,E2 -12319.491} C_VEL
LIN {X 0,Y 375.05,Z 770.427,A -85,B 0,C 180,E1 -12321.379,E2 -12321.379} C_VEL
LIN {X 0,Y 374.726,Z 775.15,A -85,B 0,C 180,E1 -12322.999,E2 -12322.999} C_VEL
LIN {X 0,Y 374.555,Z 778.763,A -85,B 0,C 180,E1 -12324.618,E2 -12324.618} C_VEL
LIN {X 0,Y 374.554,Z 780.628,A -85,B 0,C 180,E1 -12325.697,E2 -12325.697} C_VEL
LIN {X 0,Y 374.459,Z 783.023,A -85,B 0,C 180,E1 -12327.85,E2 -12327.85} C_VEL
LIN {X 0,Y 374.521,Z 784.677,A -85,B 0,C 180,E1 -12330.001,E2 -12330.001} C_VEL
LIN {X 0,Y 374.47,Z 784.753,A -85,B 0,C 180,E1 -12331.076,E2 -12331.076} C_VEL
LIN {X 0,Y 374.454,Z 784.236,A -85,B 0,C 180,E1 -12332.152,E2 -12332.152} C_VEL
LIN {X 0,Y 374.463,Z 783.119,A -85,B 0,C 180,E1 -12333.229,E2 -12333.229} C_VEL
LIN {X 0,Y 374.556,Z 781.376,A -85,B 0,C 180,E1 -12334.305,E2 -12334.305} C_VEL
LIN {X 0,Y 374.809,Z 773.69,A -85,B 0,C 180,E1 -12337.543,E2 -12337.543} C_VEL
LIN {X 0,Y 375.25,Z 767.569,A -85,B 0,C 180,E1 -12339.433,E2 -12339.433} C_VEL
LIN {X 0,Y 375.827,Z 760.886,A -85,B 0,C 180,E1 -12341.052,E2 -12341.052} C_VEL
LIN {X 0,Y 376.69,Z 752.599,A -85,B 0,C 180,E1 -12342.664,E2 -12342.664} C_VEL
LIN {X 0,Y 377.523,Z 744.102,A -85,B 0,C 180,E1 -12344.006,E2 -12344.006} C_VEL
LIN {X 0,Y 378.5,Z 733.605,A -85,B 0,C 180,E1 -12345.344,E2 -12345.344} C_VEL
LIN {X 0,Y 379.592,Z 721.789,A -85,B 0,C 180,E1 -12346.54,E2 -12346.54} C_VEL
LIN {X 0,Y 380.639,Z 709.912,A -85,B 0,C 180,E1 -12347.461,E2 -12347.461} C_VEL
LIN {X 0,Y 381.439,Z 697.55,A -85,B 0,C 180,E1 -12348.185,E2 -12348.185} C_VEL
LIN {X 0,Y 382.21,Z 684.838,A -85,B 0,C 180,E1 -12348.702,E2 -12348.702} C_VEL
LIN {X 0,Y 382.598,Z 669.684,A -85,B 0,C 180,E1 -12349.065,E2 -12349.065} C_VEL
LIN {X 0,Y 383.368,Z 601.356,A -85,B 0,C 180,E1 -12350.356,E2 -12350.356} C_VEL
LIN {X 0,Y 378.464,Z 571.824,A -85,B 0,C 180,E1 -12351.232,E2 -12351.232} C_VEL
LIN {X 0,Y 378.453,Z 570.764,A -85,B 0,C 180,E1 -12351.375,E2 -12351.375} C_VEL
LIN {X 0,Y 379.718,Z 557.08,A -85,B 0,C 180,E1 -12354.443,E2 -12354.443} C_VEL
LIN {X 0,Y 378.625,Z 550.066,A -85,B 0,C 180,E1 -12356.159,E2 -12356.159} C_VEL
LIN {X 0,Y 376.572,Z 540.019,A -85,B 0,C 180,E1 -12358.697,E2 -12358.697} C_VEL
LIN {X 0,Y 375.993,Z 537.682,A -85,B 0,C 180,E1 -12359.385,E2 -12359.385} C_VEL
LIN {X 0,Y 375.953,Z 537.656,A -85,B 0,C 180,E1 -12362.829,E2 -12362.829} C_VEL
LIN {X 0,Y 375.961,Z 537.652,A -85,B 0,C 180,E1 -12365.416,E2 -12365.416} C_VEL
LIN {X 0,Y 375.978,Z 537.652,A -85,B 0,C 180,E1 -12368.271,E2 -12368.271} C_VEL
LIN {X 0,Y 375.938,Z 537.658,A -85,B 0,C 180,E1 -12371.601,E2 -12371.601} C_VEL
LIN {X 0,Y 375.931,Z 537.659,A -85,B 0,C 180,E1 -12375.269,E2 -12375.269} C_VEL
LIN {X 0,Y 375.938,Z 537.658,A -85,B 0,C 180,E1 -12378.4,E2 -12378.4} C_VEL
LIN {X 0,Y 375.979,Z 537.654,A -85,B 0,C 180,E1 -12381.73,E2 -12381.73} C_VEL
LIN {X 0,Y 375.984,Z 537.653,A -85,B 0,C 180,E1 -12385.333,E2 -12385.333} C_VEL
LIN {X 0,Y 376.022,Z 537.967,A -85,B 0,C 180,E1 -12386.077,E2 -12386.077} C_VEL
LIN {X 0,Y 379.751,Z 548.896,A -85,B 0,C 180,E1 -12388.789,E2 -12388.789} C_VEL
LIN {X 0,Y 382.269,Z 558.402,A -85,B 0,C 180,E1 -12390.878,E2 -12390.878} C_VEL
LIN {X 0,Y 383.243,Z 564.445,A -85,B 0,C 180,E1 -12392.089,E2 -12392.089} C_VEL
LIN {X 0,Y 382.267,Z 577.036,A -85,B 0,C 180,E1 -12394.273,E2 -12394.273} C_VEL
LIN {X 0,Y 380.612,Z 599.661,A -85,B 0,C 180,E1 -12398.118,E2 -12398.118} C_VEL
LIN {X 0,Y 379.17,Z 621.968,A -85,B 0,C 180,E1 -12401.913,E2 -12401.913} C_VEL
LIN {X 0,Y 378.642,Z 632.106,A -85,B 0,C 180,E1 -12403.592,E2 -12403.592} C_VEL
LIN {X 0,Y 380.832,Z 646.384,A -85,B 0,C 180,E1 -12404.175,E2 -12404.175} C_VEL
LIN {X 0,Y 381.186,Z 651.805,A -85,B 0,C 180,E1 -12404.353,E2 -12404.353} C_VEL
LIN {X 0,Y 379.648,Z 705.157,A -85,B 0,C 180,E1 -12405.767,E2 -12405.767} C_VEL
LIN {X 0,Y 379.203,Z 715.103,A -85,B 0,C 180,E1 -12406.195,E2 -12406.195} C_VEL
LIN {X 0,Y 378.643,Z 725.906,A -85,B 0,C 180,E1 -12406.858,E2 -12406.858} C_VEL
LIN {X 0,Y 377.966,Z 735.349,A -85,B 0,C 180,E1 -12407.653,E2 -12407.653} C_VEL
LIN {X 0,Y 377.36,Z 744.106,A -85,B 0,C 180,E1 -12408.587,E2 -12408.587} C_VEL
LIN {X 0,Y 376.615,Z 752.944,A -85,B 0,C 180,E1 -12409.789,E2 -12409.789} C_VEL
LIN {X 0,Y 376.016,Z 759.195,A -85,B 0,C 180,E1 -12410.859,E2 -12410.859} C_VEL
LIN {X 0,Y 375.632,Z 764.325,A -85,B 0,C 180,E1 -12411.933,E2 -12411.933} C_VEL
LIN {X 0,Y 375.282,Z 768.515,A -85,B 0,C 180,E1 -12413.004,E2 -12413.004} C_VEL
LIN {X 0,Y 375.114,Z 771.926,A -85,B 0,C 180,E1 -12414.085,E2 -12414.085} C_VEL
LIN {X 0,Y 374.795,Z 774.614,A -85,B 0,C 180,E1 -12415.16,E2 -12415.16} C_VEL
LIN {X 0,Y 374.683,Z 775.772,A -85,B 0,C 180,E1 -12415.697,E2 -12415.697} C_VEL
LIN {X 0,Y 374.557,Z 777.466,A -85,B 0,C 180,E1 -12416.773,E2 -12416.773} C_VEL
LIN {X 0,Y 374.503,Z 778.55,A -85,B 0,C 180,E1 -12417.849,E2 -12417.849} C_VEL
LIN {X 0,Y 374.462,Z 779.056,A -85,B 0,C 180,E1 -12418.925,E2 -12418.925} C_VEL
LIN {X 0,Y 374.473,Z 778.982,A -85,B 0,C 180,E1 -12420,E2 -12420} C_VEL
LIN {X 0,Y 374.459,Z 778.328,A -85,B 0,C 180,E1 -12421.075,E2 -12421.075} C_VEL
LIN {X 0,Y 374.47,Z 777.083,A -85,B 0,C 180,E1 -12422.151,E2 -12422.151} C_VEL
LIN {X 0,Y 374.58,Z 774.038,A -85,B 0,C 180,E1 -12423.765,E2 -12423.765} C_VEL
LIN {X 0,Y 374.722,Z 769.474,A -85,B 0,C 180,E1 -12425.381,E2 -12425.381} C_VEL
LIN {X 0,Y 374.929,Z 764.259,A -85,B 0,C 180,E1 -12426.728,E2 -12426.728} C_VEL
LIN {X 0,Y 375.196,Z 759.06,A -85,B 0,C 180,E1 -12427.805,E2 -12427.805} C_VEL
LIN {X 0,Y 375.564,Z 750.956,A -85,B 0,C 180,E1 -12429.153,E2 -12429.153} C_VEL
LIN {X 0,Y 376,Z 742.534,A -85,B 0,C 180,E1 -12430.228,E2 -12430.228} C_VEL
LIN {X 0,Y 376.505,Z 733.326,A -85,B 0,C 180,E1 -12431.167,E2 -12431.167} C_VEL
LIN {X 0,Y 376.908,Z 722.809,A -85,B 0,C 180,E1 -12431.973,E2 -12431.973} C_VEL
LIN {X 0,Y 377.186,Z 713.309,A -85,B 0,C 180,E1 -12432.51,E2 -12432.51} C_VEL
LIN {X 0,Y 377.504,Z 702.233,A -85,B 0,C 180,E1 -12432.943,E2 -12432.943} C_VEL
LIN {X 0,Y 378.204,Z 647.85,A -85,B 0,C 180,E1 -12434.256,E2 -12434.256} C_VEL
LIN {X 0,Y 376.731,Z 631.747,A -85,B 0,C 180,E1 -12434.709,E2 -12434.709} C_VEL
LIN {X 0,Y 377.595,Z 610.777,A -85,B 0,C 180,E1 -12438.194,E2 -12438.194} C_VEL
LIN {X 0,Y 378.598,Z 591.065,A -85,B 0,C 180,E1 -12441.508,E2 -12441.508} C_VEL
LIN {X 0,Y 379.906,Z 567.509,A -85,B 0,C 180,E1 -12445.475,E2 -12445.475} C_VEL
LIN {X 0,Y 380.336,Z 559.024,A -85,B 0,C 180,E1 -12446.918,E2 -12446.918} C_VEL
LIN {X 0,Y 378.651,Z 549.992,A -85,B 0,C 180,E1 -12448.551,E2 -12448.551} C_VEL
LIN {X 0,Y 376.01,Z 537.78,A -85,B 0,C 180,E1 -12450.847,E2 -12450.847} C_VEL
LIN {X 0,Y 375.985,Z 537.653,A -85,B 0,C 180,E1 -12454.667,E2 -12454.667} C_VEL
LIN {X 0,Y 375.98,Z 537.653,A -85,B 0,C 180,E1 -12458.271,E2 -12458.271} C_VEL
LIN {X 0,Y 375.938,Z 537.632,A -85,B 0,C 180,E1 -12461.6,E2 -12461.6} C_VEL
LIN {X 0,Y 375.959,Z 537.648,A -85,B 0,C 180,E1 -12465.264,E2 -12465.264} C_VEL
LIN {X 0,Y 375.945,Z 537.649,A -85,B 0,C 180,E1 -12468.398,E2 -12468.398} C_VEL
LIN {X 0,Y 375.977,Z 537.64,A -85,B 0,C 180,E1 -12471.729,E2 -12471.729} C_VEL
LIN {X 0,Y 375.984,Z 537.64,A -85,B 0,C 180,E1 -12475.332,E2 -12475.332} C_VEL
LIN {X 0,Y 375.962,Z 537.65,A -85,B 0,C 180,E1 -12478.438,E2 -12478.438} C_VEL
LIN {X 0,Y 375.988,Z 537.65,A -85,B 0,C 180,E1 -12482.14,E2 -12482.14} C_VEL
LIN {X 0,Y 376.058,Z 537.746,A -85,B 0,C 180,E1 -12484.838,E2 -12484.838} C_VEL
LIN {X 0,Y 378.098,Z 548.252,A -85,B 0,C 180,E1 -12487.888,E2 -12487.888} C_VEL
LIN {X 0,Y 378.645,Z 551.771,A -85,B 0,C 180,E1 -12488.803,E2 -12488.803} C_VEL
LIN {X 0,Y 380.085,Z 557.763,A -85,B 0,C 180,E1 -12489.051,E2 -12489.051} C_VEL
LIN {X 0,Y 383.698,Z 575.591,A -85,B 0,C 180,E1 -12489.609,E2 -12489.609} C_VEL
LIN {X 0,Y 383.437,Z 607.053,A -85,B 0,C 180,E1 -12490.21,E2 -12490.21} C_VEL
LIN {X 0,Y 382.54,Z 659.152,A -85,B 0,C 180,E1 -12491.21,E2 -12491.21} C_VEL
LIN {X 0,Y 382.024,Z 672.965,A -85,B 0,C 180,E1 -12491.705,E2 -12491.705} C_VEL
LIN {X 0,Y 381.308,Z 685.331,A -85,B 0,C 180,E1 -12492.363,E2 -12492.363} C_VEL
LIN {X 0,Y 380.443,Z 697.157,A -85,B 0,C 180,E1 -12493.222,E2 -12493.222} C_VEL
LIN {X 0,Y 379.528,Z 708.526,A -85,B 0,C 180,E1 -12494.287,E2 -12494.287} C_VEL
LIN {X 0,Y 378.672,Z 718.743,A -85,B 0,C 180,E1 -12495.489,E2 -12495.489} C_VEL
LIN {X 0,Y 377.67,Z 727.923,A -85,B 0,C 180,E1 -12496.822,E2 -12496.822} C_VEL
LIN {X 0,Y 376.741,Z 736.836,A -85,B 0,C 180,E1 -12498.431,E2 -12498.431} C_VEL
LIN {X 0,Y 376.016,Z 744.008,A -85,B 0,C 180,E1 -12500.043,E2 -12500.043} C_VEL
LIN {X 0,Y 375.45,Z 748.849,A -85,B 0,C 180,E1 -12501.387,E2 -12501.387} C_VEL
LIN {X 0,Y 375.047,Z 754.305,A -85,B 0,C 180,E1 -12503.301,E2 -12503.301} C_VEL
LIN {X 0,Y 374.881,Z 757.138,A -85,B 0,C 180,E1 -12504.62,E2 -12504.62} C_VEL
LIN {X 0,Y 374.685,Z 758.998,A -85,B 0,C 180,E1 -12505.696,E2 -12505.696} C_VEL
LIN {X 0,Y 374.587,Z 760.398,A -85,B 0,C 180,E1 -12506.772,E2 -12506.772} C_VEL
LIN {X 0,Y 374.544,Z 761.652,A -85,B 0,C 180,E1 -12508.303,E2 -12508.303} C_VEL
LIN {X 0,Y 374.555,Z 762.239,A -85,B 0,C 180,E1 -12509.999,E2 -12509.999} C_VEL
LIN {X 0,Y 374.546,Z 762.051,A -85,B 0,C 180,E1 -12511.074,E2 -12511.074} C_VEL
LIN {X 0,Y 374.566,Z 760.735,A -85,B 0,C 180,E1 -12512.969,E2 -12512.969} C_VEL
LIN {X 0,Y 373.961,Z 759.809,A -85,B 0,C 180,E1 -12513.857,E2 -12513.857} C_VEL
LIN {X 0,Y 371.266,Z 757.729,A -85,B 0,C 180,E1 -12515.29,E2 -12515.29} C_VEL
LIN {X 0,Y 369.032,Z 755.559,A -85,B 0,C 180,E1 -12516.427,E2 -12516.427} C_VEL
LIN {X 0,Y 368.158,Z 753.605,A -85,B 0,C 180,E1 -12517.288,E2 -12517.288} C_VEL
LIN {X 0,Y 368.134,Z 752.863,A -85,B 0,C 180,E1 -12517.575,E2 -12517.575} C_VEL
LIN {X 0,Y 368.64,Z 747.587,A -85,B 0,C 180,E1 -12519.325,E2 -12519.325} C_VEL
LIN {X 0,Y 369.3,Z 741.276,A -85,B 0,C 180,E1 -12520.97,E2 -12520.97} C_VEL
LIN {X 0,Y 370.151,Z 733.371,A -85,B 0,C 180,E1 -12522.611,E2 -12522.611} C_VEL
LIN {X 0,Y 371.093,Z 725.312,A -85,B 0,C 180,E1 -12523.972,E2 -12523.972} C_VEL
LIN {X 0,Y 372.144,Z 715.475,A -85,B 0,C 180,E1 -12525.33,E2 -12525.33} C_VEL
LIN {X 0,Y 372.925,Z 705.803,A -85,B 0,C 180,E1 -12526.419,E2 -12526.419} C_VEL
LIN {X 0,Y 373.887,Z 695.324,A -85,B 0,C 180,E1 -12527.361,E2 -12527.361} C_VEL
LIN {X 0,Y 374.831,Z 682.691,A -85,B 0,C 180,E1 -12528.232,E2 -12528.232} C_VEL
LIN {X 0,Y 375.488,Z 670.056,A -85,B 0,C 180,E1 -12528.871,E2 -12528.871} C_VEL
LIN {X 0,Y 375.981,Z 658.066,A -85,B 0,C 180,E1 -12529.27,E2 -12529.27} C_VEL
LIN {X 0,Y 377.198,Z 577.522,A -85,B 0,C 180,E1 -12530.826,E2 -12530.826} C_VEL
LIN {X 0,Y 372.812,Z 556.078,A -85,B 0,C 180,E1 -12531.52,E2 -12531.52} C_VEL
LIN {X 0,Y 371.596,Z 551.977,A -85,B 0,C 180,E1 -12531.722,E2 -12531.722} C_VEL
LIN {X 0,Y 369.888,Z 543.118,A -85,B 0,C 180,E1 -12534.214,E2 -12534.214} C_VEL
LIN {X 0,Y 369.006,Z 538.552,A -85,B 0,C 180,E1 -12535.637,E2 -12535.637} C_VEL
LIN {X 0,Y 368.946,Z 538.515,A -85,B 0,C 180,E1 -12538.806,E2 -12538.806} C_VEL
LIN {X 0,Y 368.897,Z 538.531,A -85,B 0,C 180,E1 -12542.237,E2 -12542.237} C_VEL
LIN {X 0,Y 368.927,Z 538.531,A -85,B 0,C 180,E1 -12545,E2 -12545} C_VEL
LIN {X 0,Y 368.908,Z 538.53,A -85,B 0,C 180,E1 -12548.64,E2 -12548.64} C_VEL
LIN {X 0,Y 368.884,Z 538.535,A -85,B 0,C 180,E1 -12552.01,E2 -12552.01} C_VEL
LIN {X 0,Y 368.877,Z 538.522,A -85,B 0,C 180,E1 -12555.175,E2 -12555.175} C_VEL
LIN {X 0,Y 368.905,Z 538.53,A -85,B 0,C 180,E1 -12558.18,E2 -12558.18} C_VEL
LIN {X 0,Y 368.908,Z 538.512,A -85,B 0,C 180,E1 -12561.358,E2 -12561.358} C_VEL
LIN {X 0,Y 368.938,Z 538.529,A -85,B 0,C 180,E1 -12565.146,E2 -12565.146} C_VEL
LIN {X 0,Y 368.923,Z 538.528,A -85,B 0,C 180,E1 -12569.046,E2 -12569.046} C_VEL
LIN {X 0,Y 368.98,Z 538.518,A -85,B 0,C 180,E1 -12571.564,E2 -12571.564} C_VEL
LIN {X 0,Y 368.951,Z 538.528,A -85,B 0,C 180,E1 -12575.224,E2 -12575.224} C_VEL
LIN {X 0,Y 368.93,Z 538.521,A -85,B 0,C 180,E1 -12578.973,E2 -12578.973} C_VEL
LIN {X 0,Y 368.983,Z 538.516,A -85,B 0,C 180,E1 -12582.257,E2 -12582.257} C_VEL
LIN {X 0,Y 369.029,Z 538.514,A -85,B 0,C 180,E1 -12586.227,E2 -12586.227} C_VEL
LIN {X 0,Y 369.06,Z 538.501,A -85,B 0,C 180,E1 -12590.131,E2 -12590.131} C_VEL
LIN {X 0,Y 369.18,Z 538.495,A -85,B 0,C 180,E1 -12592.342,E2 -12592.342} C_VEL
LIN {X 0,Y 369.138,Z 538.5,A -85,B 0,C 180,E1 -12594.537,E2 -12594.537} C_VEL
LIN {X 0,Y 369.311,Z 538.475,A -85,B 0,C 180,E1 -12597.819,E2 -12597.819} C_VEL
LIN {X 0,Y 369.453,Z 538.464,A -85,B 0,C 180,E1 -12600,E2 -12600} C_VEL
LIN {X 0,Y 369.312,Z 538.474,A -85,B 0,C 180,E1 -12602.181,E2 -12602.181} C_VEL
LIN {X 0,Y 369.205,Z 538.492,A -85,B 0,C 180,E1 -12606.558,E2 -12606.558} C_VEL
LIN {X 0,Y 369.13,Z 538.499,A -85,B 0,C 180,E1 -12608.761,E2 -12608.761} C_VEL
LIN {X 0,Y 369.005,Z 538.518,A -85,B 0,C 180,E1 -12612.093,E2 -12612.093} C_VEL
LIN {X 0,Y 368.991,Z 538.515,A -85,B 0,C 180,E1 -12615.465,E2 -12615.465} C_VEL
LIN {X 0,Y 368.982,Z 538.521,A -85,B 0,C 180,E1 -12618.893,E2 -12618.893} C_VEL
LIN {X 0,Y 368.93,Z 538.523,A -85,B 0,C 180,E1 -12622.395,E2 -12622.395} C_VEL
LIN {X 0,Y 368.993,Z 538.515,A -85,B 0,C 180,E1 -12625.981,E2 -12625.981} C_VEL
LIN {X 0,Y 368.908,Z 538.532,A -85,B 0,C 180,E1 -12629.691,E2 -12629.691} C_VEL
LIN {X 0,Y 368.892,Z 538.533,A -85,B 0,C 180,E1 -12633.044,E2 -12633.044} C_VEL
LIN {X 0,Y 368.912,Z 538.511,A -85,B 0,C 180,E1 -12636.197,E2 -12636.197} C_VEL
LIN {X 0,Y 368.899,Z 538.53,A -85,B 0,C 180,E1 -12638.954,E2 -12638.954} C_VEL
LIN {X 0,Y 368.876,Z 538.523,A -85,B 0,C 180,E1 -12642.01,E2 -12642.01} C_VEL
LIN {X 0,Y 368.949,Z 538.527,A -85,B 0,C 180,E1 -12645.188,E2 -12645.188} C_VEL
LIN {X 0,Y 368.937,Z 538.529,A -85,B 0,C 180,E1 -12648.187,E2 -12648.187} C_VEL
LIN {X 0,Y 368.909,Z 538.511,A -85,B 0,C 180,E1 -12651.36,E2 -12651.36} C_VEL
LIN {X 0,Y 368.934,Z 538.531,A -85,B 0,C 180,E1 -12655.148,E2 -12655.148} C_VEL
LIN {X 0,Y 368.909,Z 538.468,A -85,B 0,C 180,E1 -12659.046,E2 -12659.046} C_VEL
LIN {X 0,Y 368.959,Z 538.669,A -85,B 0,C 180,E1 -12660.315,E2 -12660.315} C_VEL
LIN {X 0,Y 371.141,Z 548.641,A -85,B 0,C 180,E1 -12662.971,E2 -12662.971} C_VEL
LIN {X 0,Y 372.685,Z 556.914,A -85,B 0,C 180,E1 -12665.059,E2 -12665.059} C_VEL
LIN {X 0,Y 372.554,Z 561.233,A -85,B 0,C 180,E1 -12666.074,E2 -12666.074} C_VEL
LIN {X 0,Y 371.598,Z 571.302,A -85,B 0,C 180,E1 -12668.324,E2 -12668.324} C_VEL
LIN {X 0,Y 376.032,Z 597.58,A -85,B 0,C 180,E1 -12669.147,E2 -12669.147} C_VEL
LIN {X 0,Y 376.902,Z 604.244,A -85,B 0,C 180,E1 -12669.33,E2 -12669.33} C_VEL
LIN {X 0,Y 375.697,Z 679.415,A -85,B 0,C 180,E1 -12670.786,E2 -12670.786} C_VEL
LIN {X 0,Y 375.009,Z 692.618,A -85,B 0,C 180,E1 -12671.246,E2 -12671.246} C_VEL
LIN {X 0,Y 374.234,Z 704.752,A -85,B 0,C 180,E1 -12671.879,E2 -12671.879} C_VEL
LIN {X 0,Y 373.244,Z 717.008,A -85,B 0,C 180,E1 -12672.75,E2 -12672.75} C_VEL
LIN {X 0,Y 372.151,Z 728.593,A -85,B 0,C 180,E1 -12673.827,E2 -12673.827} C_VEL
LIN {X 0,Y 371.092,Z 739.381,A -85,B 0,C 180,E1 -12675.094,E2 -12675.094} C_VEL
LIN {X 0,Y 370.142,Z 749.239,A -85,B 0,C 180,E1 -12676.551,E2 -12676.551} C_VEL
LIN {X 0,Y 369.079,Z 758.171,A -85,B 0,C 180,E1 -12678.189,E2 -12678.189} C_VEL
LIN {X 0,Y 368.399,Z 765.367,A -85,B 0,C 180,E1 -12679.837,E2 -12679.837} C_VEL
LIN {X 0,Y 367.873,Z 771.919,A -85,B 0,C 180,E1 -12681.763,E2 -12681.763} C_VEL
LIN {X 0,Y 367.563,Z 776.258,A -85,B 0,C 180,E1 -12683.413,E2 -12683.413} C_VEL
LIN {X 0,Y 367.466,Z 778.558,A -85,B 0,C 180,E1 -12684.514,E2 -12684.514} C_VEL
LIN {X 0,Y 367.459,Z 780.423,A -85,B 0,C 180,E1 -12685.613,E2 -12685.613} C_VEL
LIN {X 0,Y 367.36,Z 782.818,A -85,B 0,C 180,E1 -12687.808,E2 -12687.808} C_VEL
LIN {X 0,Y 367.421,Z 784.583,A -85,B 0,C 180,E1 -12690.001,E2 -12690.001} C_VEL
LIN {X 0,Y 367.369,Z 784.73,A -85,B 0,C 180,E1 -12691.097,E2 -12691.097} C_VEL
LIN {X 0,Y 367.356,Z 784.285,A -85,B 0,C 180,E1 -12692.194,E2 -12692.194} C_VEL
LIN {X 0,Y 367.381,Z 783.221,A -85,B 0,C 180,E1 -12693.291,E2 -12693.291} C_VEL
LIN {X 0,Y 367.484,Z 781.524,A -85,B 0,C 180,E1 -12694.388,E2 -12694.388} C_VEL
LIN {X 0,Y 367.515,Z 777.661,A -85,B 0,C 180,E1 -12696.066,E2 -12696.066} C_VEL
LIN {X 0,Y 367.875,Z 771.888,A -85,B 0,C 180,E1 -12698.239,E2 -12698.239} C_VEL
LIN {X 0,Y 368.312,Z 766.349,A -85,B 0,C 180,E1 -12699.89,E2 -12699.89} C_VEL
LIN {X 0,Y 368.964,Z 759.441,A -85,B 0,C 180,E1 -12701.538,E2 -12701.538} C_VEL
LIN {X 0,Y 369.922,Z 750.802,A -85,B 0,C 180,E1 -12703.179,E2 -12703.179} C_VEL
LIN {X 0,Y 370.802,Z 742.089,A -85,B 0,C 180,E1 -12704.525,E2 -12704.525} C_VEL
LIN {X 0,Y 371.761,Z 732.22,A -85,B 0,C 180,E1 -12705.77,E2 -12705.77} C_VEL
LIN {X 0,Y 372.784,Z 721.58,A -85,B 0,C 180,E1 -12706.851,E2 -12706.851} C_VEL
LIN {X 0,Y 373.866,Z 709.702,A -85,B 0,C 180,E1 -12707.787,E2 -12707.787} C_VEL
LIN {X 0,Y 374.697,Z 697.338,A -85,B 0,C 180,E1 -12708.524,E2 -12708.524} C_VEL
LIN {X 0,Y 375.495,Z 684.623,A -85,B 0,C 180,E1 -12709.05,E2 -12709.05} C_VEL
LIN {X 0,Y 375.858,Z 671.249,A -85,B 0,C 180,E1 -12709.385,E2 -12709.385} C_VEL
LIN {X 0,Y 376.731,Z 602.273,A -85,B 0,C 180,E1 -12710.708,E2 -12710.708} C_VEL
LIN {X 0,Y 371.789,Z 572.691,A -85,B 0,C 180,E1 -12711.595,E2 -12711.595} C_VEL
LIN {X 0,Y 371.581,Z 570.939,A -85,B 0,C 180,E1 -12711.716,E2 -12711.716} C_VEL
LIN {X 0,Y 372.765,Z 558.653,A -85,B 0,C 180,E1 -12714.506,E2 -12714.506} C_VEL
LIN {X 0,Y 371.867,Z 552.375,A -85,B 0,C 180,E1 -12716.067,E2 -12716.067} C_VEL
LIN {X 0,Y 369.757,Z 541.888,A -85,B 0,C 180,E1 -12718.771,E2 -12718.771} C_VEL
LIN {X 0,Y 368.957,Z 538.564,A -85,B 0,C 180,E1 -12719.727,E2 -12719.727} C_VEL
LIN {X 0,Y 368.9,Z 538.532,A -85,B 0,C 180,E1 -12723.539,E2 -12723.539} C_VEL
LIN {X 0,Y 368.905,Z 538.53,A -85,B 0,C 180,E1 -12726.856,E2 -12726.856} C_VEL
LIN {X 0,Y 368.914,Z 538.53,A -85,B 0,C 180,E1 -12730.371,E2 -12730.371} C_VEL
LIN {X 0,Y 368.887,Z 538.537,A -85,B 0,C 180,E1 -12733.616,E2 -12733.616} C_VEL
LIN {X 0,Y 368.889,Z 538.536,A -85,B 0,C 180,E1 -12736.696,E2 -12736.696} C_VEL
LIN {X 0,Y 368.915,Z 538.531,A -85,B 0,C 180,E1 -12739.643,E2 -12739.643} C_VEL
LIN {X 0,Y 368.907,Z 538.535,A -85,B 0,C 180,E1 -12743.144,E2 -12743.144} C_VEL
LIN {X 0,Y 368.961,Z 538.788,A -85,B 0,C 180,E1 -12745.054,E2 -12745.054} C_VEL
LIN {X 0,Y 372.914,Z 549.816,A -85,B 0,C 180,E1 -12748.004,E2 -12748.004} C_VEL
LIN {X 0,Y 375.338,Z 558.514,A -85,B 0,C 180,E1 -12750.036,E2 -12750.036} C_VEL
LIN {X 0,Y 376.787,Z 566.353,A -85,B 0,C 180,E1 -12751.701,E2 -12751.701} C_VEL
LIN {X 0,Y 376.294,Z 573.958,A -85,B 0,C 180,E1 -12753.069,E2 -12753.069} C_VEL
LIN {X 0,Y 374.476,Z 595.831,A -85,B 0,C 180,E1 -12756.87,E2 -12756.87} C_VEL
LIN {X 0,Y 372.795,Z 618.409,A -85,B 0,C 180,E1 -12760.766,E2 -12760.766} C_VEL
LIN {X 0,Y 371.976,Z 632.145,A -85,B 0,C 180,E1 -12763.091,E2 -12763.091} C_VEL
LIN {X 0,Y 374.311,Z 646.607,A -85,B 0,C 180,E1 -12763.723,E2 -12763.723} C_VEL
LIN {X 0,Y 374.713,Z 651.794,A -85,B 0,C 180,E1 -12763.91,E2 -12763.91} C_VEL
LIN {X 0,Y 373.006,Z 705.749,A -85,B 0,C 180,E1 -12765.404,E2 -12765.404} C_VEL
LIN {X 0,Y 372.555,Z 714.879,A -85,B 0,C 180,E1 -12765.804,E2 -12765.804} C_VEL
LIN {X 0,Y 371.952,Z 725.774,A -85,B 0,C 180,E1 -12766.478,E2 -12766.478} C_VEL
LIN {X 0,Y 371.226,Z 735.265,A -85,B 0,C 180,E1 -12767.286,E2 -12767.286} C_VEL
LIN {X 0,Y 370.528,Z 744.043,A -85,B 0,C 180,E1 -12768.235,E2 -12768.235} C_VEL
LIN {X 0,Y 369.791,Z 752.054,A -85,B 0,C 180,E1 -12769.321,E2 -12769.321} C_VEL
LIN {X 0,Y 369.217,Z 758.427,A -85,B 0,C 180,E1 -12770.412,E2 -12770.412} C_VEL
LIN {X 0,Y 368.623,Z 764.845,A -85,B 0,C 180,E1 -12771.779,E2 -12771.779} C_VEL
LIN {X 0,Y 368.235,Z 769.283,A -85,B 0,C 180,E1 -12772.961,E2 -12772.961} C_VEL
LIN {X 0,Y 367.91,Z 773.749,A -85,B 0,C 180,E1 -12774.519,E2 -12774.519} C_VEL
LIN {X 0,Y 367.622,Z 776.046,A -85,B 0,C 180,E1 -12775.614,E2 -12775.614} C_VEL
LIN {X 0,Y 367.474,Z 777.695,A -85,B 0,C 180,E1 -12776.711,E2 -12776.711} C_VEL
LIN {X 0,Y 367.407,Z 778.722,A -85,B 0,C 180,E1 -12777.808,E2 -12777.808} C_VEL
LIN {X 0,Y 367.363,Z 779.153,A -85,B 0,C 180,E1 -12778.904,E2 -12778.904} C_VEL
LIN {X 0,Y 367.374,Z 779.005,A -85,B 0,C 180,E1 -12780,E2 -12780} C_VEL
LIN {X 0,Y 367.359,Z 778.277,A -85,B 0,C 180,E1 -12781.096,E2 -12781.096} C_VEL
LIN {X 0,Y 367.373,Z 776.958,A -85,B 0,C 180,E1 -12782.193,E2 -12782.193} C_VEL
LIN {X 0,Y 367.506,Z 773.841,A -85,B 0,C 180,E1 -12783.838,E2 -12783.838} C_VEL
LIN {X 0,Y 367.634,Z 769.114,A -85,B 0,C 180,E1 -12785.485,E2 -12785.485} C_VEL
LIN {X 0,Y 367.893,Z 763.798,A -85,B 0,C 180,E1 -12786.857,E2 -12786.857} C_VEL
LIN {X 0,Y 368.195,Z 757.041,A -85,B 0,C 180,E1 -12788.231,E2 -12788.231} C_VEL
LIN {X 0,Y 368.583,Z 749.126,A -85,B 0,C 180,E1 -12789.466,E2 -12789.466} C_VEL
LIN {X 0,Y 369.019,Z 741.518,A -85,B 0,C 180,E1 -12790.424,E2 -12790.424} C_VEL
LIN {X 0,Y 369.457,Z 732.016,A -85,B 0,C 180,E1 -12791.383,E2 -12791.383} C_VEL
LIN {X 0,Y 369.904,Z 722.001,A -85,B 0,C 180,E1 -12792.133,E2 -12792.133} C_VEL
LIN {X 0,Y 370.13,Z 713.633,A -85,B 0,C 180,E1 -12792.613,E2 -12792.613} C_VEL
LIN {X 0,Y 370.455,Z 702.764,A -85,B 0,C 180,E1 -12793.055,E2 -12793.055} C_VEL
LIN {X 0,Y 371.184,Z 648.265,A -85,B 0,C 180,E1 -12794.41,E2 -12794.41} C_VEL
LIN {X 0,Y 369.697,Z 631.583,A -85,B 0,C 180,E1 -12794.906,E2 -12794.906} C_VEL
LIN {X 0,Y 370.601,Z 611.004,A -85,B 0,C 180,E1 -12798.383,E2 -12798.383} C_VEL
LIN {X 0,Y 371.626,Z 590.938,A -85,B 0,C 180,E1 -12801.796,E2 -12801.796} C_VEL
LIN {X 0,Y 372.961,Z 568.137,A -85,B 0,C 180,E1 -12805.684,E2 -12805.684} C_VEL
LIN {X 0,Y 373.353,Z 559.991,A -85,B 0,C 180,E1 -12807.081,E2 -12807.081} C_VEL
LIN {X 0,Y 370.708,Z 546.722,A -85,B 0,C 180,E1 -12809.533,E2 -12809.533} C_VEL
LIN {X 0,Y 368.979,Z 538.651,A -85,B 0,C 180,E1 -12811.092,E2 -12811.092} C_VEL
LIN {X 0,Y 368.934,Z 538.529,A -85,B 0,C 180,E1 -12815.001,E2 -12815.001} C_VEL
LIN {X 0,Y 368.914,Z 538.531,A -85,B 0,C 180,E1 -12818.64,E2 -12818.64} C_VEL
LIN {X 0,Y 368.885,Z 538.503,A -85,B 0,C 180,E1 -12822.009,E2 -12822.009} C_VEL
LIN {X 0,Y 368.932,Z 538.52,A -85,B 0,C 180,E1 -12825.183,E2 -12825.183} C_VEL
LIN {X 0,Y 368.893,Z 538.531,A -85,B 0,C 180,E1 -12828.178,E2 -12828.178} C_VEL
LIN {X 0,Y 368.912,Z 538.514,A -85,B 0,C 180,E1 -12831.36,E2 -12831.36} C_VEL
LIN {X 0,Y 368.941,Z 538.518,A -85,B 0,C 180,E1 -12835.146,E2 -12835.146} C_VEL
LIN {X 0,Y 368.934,Z 538.525,A -85,B 0,C 180,E1 -12839.046,E2 -12839.046} C_VEL
LIN {X 0,Y 368.967,Z 538.526,A -85,B 0,C 180,E1 -12842.796,E2 -12842.796} C_VEL
LIN {X 0,Y 369.014,Z 538.685,A -85,B 0,C 180,E1 -12844.55,E2 -12844.55} C_VEL
LIN {X 0,Y 370.917,Z 548.449,A -85,B 0,C 180,E1 -12847.437,E2 -12847.437} C_VEL
LIN {X 0,Y 371.587,Z 551.987,A -85,B 0,C 180,E1 -12848.381,E2 -12848.381} C_VEL
LIN {X 0,Y 373.1,Z 557.34,A -85,B 0,C 180,E1 -12848.626,E2 -12848.626} C_VEL
LIN {X 0,Y 377.144,Z 577.045,A -85,B 0,C 180,E1 -12849.263,E2 -12849.263} C_VEL
LIN {X 0,Y 375.87,Z 658.197,A -85,B 0,C 180,E1 -12850.828,E2 -12850.828} C_VEL
LIN {X 0,Y 375.385,Z 671.658,A -85,B 0,C 180,E1 -12851.299,E2 -12851.299} C_VEL
LIN {X 0,Y 374.649,Z 684.443,A -85,B 0,C 180,E1 -12851.969,E2 -12851.969} C_VEL
LIN {X 0,Y 373.821,Z 695.781,A -85,B 0,C 180,E1 -12852.775,E2 -12852.775} C_VEL
LIN {X 0,Y 372.832,Z 706.983,A -85,B 0,C 180,E1 -12853.806,E2 -12853.806} C_VEL
LIN {X 0,Y 371.938,Z 717.891,A -85,B 0,C 180,E1 -12855.08,E2 -12855.08} C_VEL
LIN {X 0,Y 370.964,Z 726.436,A -85,B 0,C 180,E1 -12856.3,E2 -12856.3} C_VEL
LIN {X 0,Y 370.095,Z 734.306,A -85,B 0,C 180,E1 -12857.664,E2 -12857.664} C_VEL
LIN {X 0,Y 369.244,Z 741.996,A -85,B 0,C 180,E1 -12859.304,E2 -12859.304} C_VEL
LIN {X 0,Y 368.42,Z 749.056,A -85,B 0,C 180,E1 -12861.221,E2 -12861.221} C_VEL
LIN {X 0,Y 368.042,Z 753.755,A -85,B 0,C 180,E1 -12862.87,E2 -12862.87} C_VEL
LIN {X 0,Y 367.812,Z 757.344,A -85,B 0,C 180,E1 -12864.517,E2 -12864.517} C_VEL
LIN {X 0,Y 367.62,Z 759.203,A -85,B 0,C 180,E1 -12865.613,E2 -12865.613} C_VEL
LIN {X 0,Y 367.501,Z 760.603,A -85,B 0,C 180,E1 -12866.71,E2 -12866.71} C_VEL
LIN {X 0,Y 367.45,Z 762.211,A -85,B 0,C 180,E1 -12868.903,E2 -12868.903} C_VEL
LIN {X 0,Y 367.458,Z 762.444,A -85,B 0,C 180,E1 -12869.999,E2 -12869.999} C_VEL
LIN {X 0,Y 367.45,Z 762.256,A -85,B 0,C 180,E1 -12871.095,E2 -12871.095} C_VEL
LIN {X 0,Y 367.475,Z 760.978,A -85,B 0,C 180,E1 -12872.982,E2 -12872.982} C_VEL
LIN {X 0,Y 367.612,Z 759.354,A -85,B 0,C 180,E1 -12874.385,E2 -12874.385} C_VEL
LIN {X 0,Y 367.887,Z 756.023,A -85,B 0,C 180,E1 -12876.254,E2 -12876.254} C_VEL
LIN {X 0,Y 368.134,Z 752.863,A -85,B 0,C 180,E1 -12877.575,E2 -12877.575} C_VEL
LIN {X 0,Y 367.672,Z 750.59,A -85,B 0,C 180,E1 -12878.423,E2 -12878.423} C_VEL
LIN {X 0,Y 365.254,Z 746.478,A -85,B 0,C 180,E1 -12879.785,E2 -12879.785} C_VEL
LIN {X 0,Y 362.964,Z 741.7,A -85,B 0,C 180,E1 -12881.107,E2 -12881.107} C_VEL
LIN {X 0,Y 362.706,Z 738.382,A -85,B 0,C 180,E1 -12881.88,E2 -12881.88} C_VEL
LIN {X 0,Y 363.578,Z 730.547,A -85,B 0,C 180,E1 -12883.411,E2 -12883.411} C_VEL
LIN {X 0,Y 364.673,Z 721.82,A -85,B 0,C 180,E1 -12884.793,E2 -12884.793} C_VEL
LIN {X 0,Y 365.548,Z 712.661,A -85,B 0,C 180,E1 -12885.992,E2 -12885.992} C_VEL
LIN {X 0,Y 366.543,Z 701.773,A -85,B 0,C 180,E1 -12887.144,E2 -12887.144} C_VEL
LIN {X 0,Y 367.571,Z 690.162,A -85,B 0,C 180,E1 -12888.1,E2 -12888.1} C_VEL
LIN {X 0,Y 368.43,Z 678.08,A -85,B 0,C 180,E1 -12888.849,E2 -12888.849} C_VEL
LIN {X 0,Y 368.974,Z 665.829,A -85,B 0,C 180,E1 -12889.397,E2 -12889.397} C_VEL
LIN {X 0,Y 369.393,Z 653.764,A -85,B 0,C 180,E1 -12889.736,E2 -12889.736} C_VEL
LIN {X 0,Y 370.506,Z 577.839,A -85,B 0,C 180,E1 -12891.217,E2 -12891.217} C_VEL
LIN {X 0,Y 366.301,Z 557.772,A -85,B 0,C 180,E1 -12891.89,E2 -12891.89} C_VEL
LIN {X 0,Y 364.487,Z 552.246,A -85,B 0,C 180,E1 -12892.162,E2 -12892.162} C_VEL
LIN {X 0,Y 362.692,Z 543.207,A -85,B 0,C 180,E1 -12894.76,E2 -12894.76} C_VEL
LIN {X 0,Y 361.974,Z 539.422,A -85,B 0,C 180,E1 -12895.979,E2 -12895.979} C_VEL
LIN {X 0,Y 361.892,Z 539.391,A -85,B 0,C 180,E1 -12899.084,E2 -12899.084} C_VEL
LIN {X 0,Y 361.847,Z 539.408,A -85,B 0,C 180,E1 -12902.943,E2 -12902.943} C_VEL
LIN {X 0,Y 361.866,Z 539.404,A -85,B 0,C 180,E1 -12905.635,E2 -12905.635} C_VEL
LIN {X 0,Y 361.87,Z 539.404,A -85,B 0,C 180,E1 -12909.026,E2 -12909.026} C_VEL
LIN {X 0,Y 361.834,Z 539.413,A -85,B 0,C 180,E1 -12912.827,E2 -12912.827} C_VEL
LIN {X 0,Y 361.822,Z 539.407,A -85,B 0,C 180,E1 -12915.944,E2 -12915.944} C_VEL
LIN {X 0,Y 361.868,Z 539.405,A -85,B 0,C 180,E1 -12919.237,E2 -12919.237} C_VEL
LIN {X 0,Y 361.869,Z 539.396,A -85,B 0,C 180,E1 -12922.982,E2 -12922.982} C_VEL
LIN {X 0,Y 361.857,Z 539.407,A -85,B 0,C 180,E1 -12926.629,E2 -12926.629} C_VEL
LIN {X 0,Y 361.87,Z 539.411,A -85,B 0,C 180,E1 -12929.671,E2 -12929.671} C_VEL
LIN {X 0,Y 361.948,Z 539.395,A -85,B 0,C 180,E1 -12933.474,E2 -12933.474} C_VEL
LIN {X 0,Y 361.884,Z 539.402,A -85,B 0,C 180,E1 -12937.144,E2 -12937.144} C_VEL
LIN {X 0,Y 361.915,Z 539.4,A -85,B 0,C 180,E1 -12940.724,E2 -12940.724} C_VEL
LIN {X 0,Y 361.938,Z 539.39,A -85,B 0,C 180,E1 -12944.226,E2 -12944.226} C_VEL
LIN {X 0,Y 361.991,Z 539.39,A -85,B 0,C 180,E1 -12946.527,E2 -12946.527} C_VEL
LIN {X 0,Y 362.024,Z 539.377,A -85,B 0,C 180,E1 -12949.938,E2 -12949.938} C_VEL
LIN {X 0,Y 362.143,Z 539.372,A -85,B 0,C 180,E1 -12952.192,E2 -12952.192} C_VEL
LIN {X 0,Y 362.111,Z 539.375,A -85,B 0,C 180,E1 -12954.431,E2 -12954.431} C_VEL
LIN {X 0,Y 362.275,Z 539.35,A -85,B 0,C 180,E1 -12957.776,E2 -12957.776} C_VEL
LIN {X 0,Y 362.422,Z 539.34,A -85,B 0,C 180,E1 -12960,E2 -12960} C_VEL
LIN {X 0,Y 362.276,Z 539.35,A -85,B 0,C 180,E1 -12962.224,E2 -12962.224} C_VEL
LIN {X 0,Y 362.168,Z 539.369,A -85,B 0,C 180,E1 -12966.686,E2 -12966.686} C_VEL
LIN {X 0,Y 362.067,Z 539.379,A -85,B 0,C 180,E1 -12968.933,E2 -12968.933} C_VEL
LIN {X 0,Y 361.959,Z 539.395,A -85,B 0,C 180,E1 -12972.332,E2 -12972.332} C_VEL
LIN {X 0,Y 361.955,Z 539.393,A -85,B 0,C 180,E1 -12974.621,E2 -12974.621} C_VEL
LIN {X 0,Y 361.953,Z 539.397,A -85,B 0,C 180,E1 -12978.1,E2 -12978.1} C_VEL
LIN {X 0,Y 361.892,Z 539.4,A -85,B 0,C 180,E1 -12981.653,E2 -12981.653} C_VEL
LIN {X 0,Y 361.921,Z 539.403,A -85,B 0,C 180,E1 -12985.291,E2 -12985.291} C_VEL
LIN {X 0,Y 361.901,Z 539.404,A -85,B 0,C 180,E1 -12987.78,E2 -12987.78} C_VEL
LIN {X 0,Y 361.832,Z 539.411,A -85,B 0,C 180,E1 -12991.63,E2 -12991.63} C_VEL
LIN {X 0,Y 361.868,Z 539.397,A -85,B 0,C 180,E1 -12995.346,E2 -12995.346} C_VEL
LIN {X 0,Y 361.865,Z 539.406,A -85,B 0,C 180,E1 -12999.028,E2 -12999.028} C_VEL
LIN {X 0,Y 361.833,Z 539.4,A -85,B 0,C 180,E1 -13002.829,E2 -13002.829} C_VEL
LIN {X 0,Y 361.894,Z 539.401,A -85,B 0,C 180,E1 -13005.934,E2 -13005.934} C_VEL
LIN {X 0,Y 361.901,Z 539.406,A -85,B 0,C 180,E1 -13009.233,E2 -13009.233} C_VEL
LIN {X 0,Y 361.866,Z 539.387,A -85,B 0,C 180,E1 -13012.983,E2 -13012.983} C_VEL
LIN {X 0,Y 361.856,Z 539.378,A -85,B 0,C 180,E1 -13016.632,E2 -13016.632} C_VEL
LIN {X 0,Y 361.918,Z 539.458,A -85,B 0,C 180,E1 -13019.903,E2 -13019.903} C_VEL
LIN {X 0,Y 364.101,Z 549.294,A -85,B 0,C 180,E1 -13022.612,E2 -13022.612} C_VEL
LIN {X 0,Y 365.793,Z 558.535,A -85,B 0,C 180,E1 -13024.997,E2 -13024.997} C_VEL
LIN {X 0,Y 365.229,Z 566.008,A -85,B 0,C 180,E1 -13026.768,E2 -13026.768} C_VEL
LIN {X 0,Y 364.777,Z 571.09,A -85,B 0,C 180,E1 -13027.896,E2 -13027.896} C_VEL
LIN {X 0,Y 369.419,Z 598.609,A -85,B 0,C 180,E1 -13028.781,E2 -13028.781} C_VEL
LIN {X 0,Y 370.26,Z 605.238,A -85,B 0,C 180,E1 -13028.966,E2 -13028.966} C_VEL
LIN {X 0,Y 369.011,Z 679.224,A -85,B 0,C 180,E1 -13030.424,E2 -13030.424} C_VEL
LIN {X 0,Y 368.297,Z 692.422,A -85,B 0,C 180,E1 -13030.891,E2 -13030.891} C_VEL
LIN {X 0,Y 367.505,Z 704.554,A -85,B 0,C 180,E1 -13031.536,E2 -13031.536} C_VEL
LIN {X 0,Y 366.451,Z 716.807,A -85,B 0,C 180,E1 -13032.42,E2 -13032.42} C_VEL
LIN {X 0,Y 365.317,Z 728.391,A -85,B 0,C 180,E1 -13033.516,E2 -13033.516} C_VEL
LIN {X 0,Y 364.187,Z 739.378,A -85,B 0,C 180,E1 -13034.832,E2 -13034.832} C_VEL
LIN {X 0,Y 363.212,Z 749.036,A -85,B 0,C 180,E1 -13036.29,E2 -13036.29} C_VEL
LIN {X 0,Y 362.114,Z 757.968,A -85,B 0,C 180,E1 -13037.959,E2 -13037.959} C_VEL
LIN {X 0,Y 361.388,Z 765.163,A -85,B 0,C 180,E1 -13039.638,E2 -13039.638} C_VEL
LIN {X 0,Y 360.817,Z 771.714,A -85,B 0,C 180,E1 -13041.601,E2 -13041.601} C_VEL
LIN {X 0,Y 360.498,Z 776.053,A -85,B 0,C 180,E1 -13043.284,E2 -13043.284} C_VEL
LIN {X 0,Y 360.382,Z 778.354,A -85,B 0,C 180,E1 -13044.405,E2 -13044.405} C_VEL
LIN {X 0,Y 360.367,Z 780.218,A -85,B 0,C 180,E1 -13045.527,E2 -13045.527} C_VEL
LIN {X 0,Y 360.301,Z 781.613,A -85,B 0,C 180,E1 -13046.646,E2 -13046.646} C_VEL
LIN {X 0,Y 360.322,Z 784.484,A -85,B 0,C 180,E1 -13050.001,E2 -13050.001} C_VEL
LIN {X 0,Y 360.267,Z 784.71,A -85,B 0,C 180,E1 -13051.119,E2 -13051.119} C_VEL
LIN {X 0,Y 360.261,Z 784.317,A -85,B 0,C 180,E1 -13052.237,E2 -13052.237} C_VEL
LIN {X 0,Y 360.303,Z 783.299,A -85,B 0,C 180,E1 -13053.356,E2 -13053.356} C_VEL
LIN {X 0,Y 360.395,Z 780.586,A -85,B 0,C 180,E1 -13055.035,E2 -13055.035} C_VEL
LIN {X 0,Y 360.445,Z 778.275,A -85,B 0,C 180,E1 -13056.063,E2 -13056.063} C_VEL
LIN {X 0,Y 360.948,Z 769.98,A -85,B 0,C 180,E1 -13058.962,E2 -13058.962} C_VEL
LIN {X 0,Y 361.608,Z 762.874,A -85,B 0,C 180,E1 -13060.924,E2 -13060.924} C_VEL
LIN {X 0,Y 362.475,Z 755.167,A -85,B 0,C 180,E1 -13062.6,E2 -13062.6} C_VEL
LIN {X 0,Y 363.496,Z 745.488,A -85,B 0,C 180,E1 -13064.272,E2 -13064.272} C_VEL
LIN {X 0,Y 364.528,Z 735.506,A -85,B 0,C 180,E1 -13065.66,E2 -13065.66} C_VEL
LIN {X 0,Y 365.682,Z 724.23,A -85,B 0,C 180,E1 -13066.9,E2 -13066.9} C_VEL
LIN {X 0,Y 366.771,Z 713.19,A -85,B 0,C 180,E1 -13067.855,E2 -13067.855} C_VEL
LIN {X 0,Y 367.731,Z 700.955,A -85,B 0,C 180,E1 -13068.671,E2 -13068.671} C_VEL
LIN {X 0,Y 368.556,Z 688.075,A -85,B 0,C 180,E1 -13069.278,E2 -13069.278} C_VEL
LIN {X 0,Y 369.07,Z 674.37,A -85,B 0,C 180,E1 -13069.684,E2 -13069.684} C_VEL
LIN {X 0,Y 370.097,Z 603.203,A -85,B 0,C 180,E1 -13071.073,E2 -13071.073} C_VEL
LIN {X 0,Y 365.18,Z 573.78,A -85,B 0,C 180,E1 -13071.976,E2 -13071.976} C_VEL
LIN {X 0,Y 364.736,Z 570.997,A -85,B 0,C 180,E1 -13072.109,E2 -13072.109} C_VEL
LIN {X 0,Y 365.836,Z 559.707,A -85,B 0,C 180,E1 -13074.699,E2 -13074.699} C_VEL
LIN {X 0,Y 364.649,Z 552.271,A -85,B 0,C 180,E1 -13076.598,E2 -13076.598} C_VEL
LIN {X 0,Y 362.813,Z 543.324,A -85,B 0,C 180,E1 -13078.966,E2 -13078.966} C_VEL
LIN {X 0,Y 361.914,Z 539.486,A -85,B 0,C 180,E1 -13080.061,E2 -13080.061} C_VEL
LIN {X 0,Y 361.858,Z 539.412,A -85,B 0,C 180,E1 -13084.281,E2 -13084.281} C_VEL
LIN {X 0,Y 361.867,Z 539.407,A -85,B 0,C 180,E1 -13087.223,E2 -13087.223} C_VEL
LIN {X 0,Y 361.839,Z 539.41,A -85,B 0,C 180,E1 -13090.756,E2 -13090.756} C_VEL
LIN {X 0,Y 361.821,Z 539.413,A -85,B 0,C 180,E1 -13094.369,E2 -13094.369} C_VEL
LIN {X 0,Y 361.84,Z 539.412,A -85,B 0,C 180,E1 -13097.568,E2 -13097.568} C_VEL
LIN {X 0,Y 361.874,Z 539.407,A -85,B 0,C 180,E1 -13100.974,E2 -13100.974} C_VEL
LIN {X 0,Y 361.907,Z 539.631,A -85,B 0,C 180,E1 -13103.874,E2 -13103.874} C_VEL
LIN {X 0,Y 364.621,Z 546.736,A -85,B 0,C 180,E1 -13106.015,E2 -13106.015} C_VEL
LIN {X 0,Y 367.646,Z 555.845,A -85,B 0,C 180,E1 -13108.431,E2 -13108.431} C_VEL
LIN {X 0,Y 369.91,Z 565.28,A -85,B 0,C 180,E1 -13110.628,E2 -13110.628} C_VEL
LIN {X 0,Y 370.477,Z 570.378,A -85,B 0,C 180,E1 -13111.689,E2 -13111.689} C_VEL
LIN {X 0,Y 368.411,Z 591.654,A -85,B 0,C 180,E1 -13115.486,E2 -13115.486} C_VEL
LIN {X 0,Y 367.093,Z 608.073,A -85,B 0,C 180,E1 -13118.374,E2 -13118.374} C_VEL
LIN {X 0,Y 365.349,Z 631.43,A -85,B 0,C 180,E1 -13122.472,E2 -13122.472} C_VEL
LIN {X 0,Y 365.519,Z 633.109,A -85,B 0,C 180,E1 -13122.624,E2 -13122.624} C_VEL
LIN {X 0,Y 367.884,Z 647.429,A -85,B 0,C 180,E1 -13123.277,E2 -13123.277} C_VEL
LIN {X 0,Y 368.211,Z 654.461,A -85,B 0,C 180,E1 -13123.521,E2 -13123.521} C_VEL
LIN {X 0,Y 366.458,Z 705.102,A -85,B 0,C 180,E1 -13124.959,E2 -13124.959} C_VEL
LIN {X 0,Y 365.944,Z 714.941,A -85,B 0,C 180,E1 -13125.4,E2 -13125.4} C_VEL
LIN {X 0,Y 365.291,Z 725.739,A -85,B 0,C 180,E1 -13126.084,E2 -13126.084} C_VEL
LIN {X 0,Y 364.503,Z 735.19,A -85,B 0,C 180,E1 -13126.906,E2 -13126.906} C_VEL
LIN {X 0,Y 363.777,Z 743.997,A -85,B 0,C 180,E1 -13127.872,E2 -13127.872} C_VEL
LIN {X 0,Y 362.871,Z 752.886,A -85,B 0,C 180,E1 -13129.115,E2 -13129.115} C_VEL
LIN {X 0,Y 362.271,Z 759.145,A -85,B 0,C 180,E1 -13130.227,E2 -13130.227} C_VEL
LIN {X 0,Y 361.714,Z 764.304,A -85,B 0,C 180,E1 -13131.339,E2 -13131.339} C_VEL
LIN {X 0,Y 361.286,Z 768.802,A -85,B 0,C 180,E1 -13132.535,E2 -13132.535} C_VEL
LIN {X 0,Y 361.045,Z 772.709,A -85,B 0,C 180,E1 -13133.854,E2 -13133.854} C_VEL
LIN {X 0,Y 360.564,Z 776.298,A -85,B 0,C 180,E1 -13135.528,E2 -13135.528} C_VEL
LIN {X 0,Y 360.394,Z 777.899,A -85,B 0,C 180,E1 -13136.646,E2 -13136.646} C_VEL
LIN {X 0,Y 360.311,Z 778.881,A -85,B 0,C 180,E1 -13137.764,E2 -13137.764} C_VEL
LIN {X 0,Y 360.265,Z 779.251,A -85,B 0,C 180,E1 -13138.882,E2 -13138.882} C_VEL
LIN {X 0,Y 360.274,Z 779.024,A -85,B 0,C 180,E1 -13140,E2 -13140} C_VEL
LIN {X 0,Y 360.258,Z 778.215,A -85,B 0,C 180,E1 -13141.118,E2 -13141.118} C_VEL
LIN {X 0,Y 360.304,Z 775.944,A -85,B 0,C 180,E1 -13142.795,E2 -13142.795} C_VEL
LIN {X 0,Y 360.495,Z 772.1,A -85,B 0,C 180,E1 -13144.473,E2 -13144.473} C_VEL
LIN {X 0,Y 360.565,Z 767.622,A -85,B 0,C 180,E1 -13145.895,E2 -13145.895} C_VEL
LIN {X 0,Y 360.915,Z 762.034,A -85,B 0,C 180,E1 -13147.272,E2 -13147.272} C_VEL
LIN {X 0,Y 361.22,Z 754.58,A -85,B 0,C 180,E1 -13148.673,E2 -13148.673} C_VEL
LIN {X 0,Y 361.669,Z 747.166,A -85,B 0,C 180,E1 -13149.79,E2 -13149.79} C_VEL
LIN {X 0,Y 362.087,Z 737.772,A -85,B 0,C 180,E1 -13150.909,E2 -13150.909} C_VEL
LIN {X 0,Y 362.504,Z 728.653,A -85,B 0,C 180,E1 -13151.746,E2 -13151.746} C_VEL
LIN {X 0,Y 362.916,Z 718.896,A -85,B 0,C 180,E1 -13152.441,E2 -13152.441} C_VEL
LIN {X 0,Y 363.28,Z 707.666,A -85,B 0,C 180,E1 -13152.997,E2 -13152.997} C_VEL
LIN {X 0,Y 363.474,Z 695.288,A -85,B 0,C 180,E1 -13153.381,E2 -13153.381} C_VEL
LIN {X 0,Y 364.269,Z 650.267,A -85,B 0,C 180,E1 -13154.526,E2 -13154.526} C_VEL
LIN {X 0,Y 362.673,Z 631.562,A -85,B 0,C 180,E1 -13155.086,E2 -13155.086} C_VEL
LIN {X 0,Y 363.608,Z 611.184,A -85,B 0,C 180,E1 -13158.578,E2 -13158.578} C_VEL
LIN {X 0,Y 364.744,Z 590.053,A -85,B 0,C 180,E1 -13162.217,E2 -13162.217} C_VEL
LIN {X 0,Y 366.028,Z 568.258,A -85,B 0,C 180,E1 -13165.979,E2 -13165.979} C_VEL
LIN {X 0,Y 366.293,Z 560.039,A -85,B 0,C 180,E1 -13167.419,E2 -13167.419} C_VEL
LIN {X 0,Y 362.776,Z 543.368,A -85,B 0,C 180,E1 -13170.553,E2 -13170.553} C_VEL
LIN {X 0,Y 361.921,Z 539.507,A -85,B 0,C 180,E1 -13171.352,E2 -13171.352} C_VEL
LIN {X 0,Y 361.879,Z 539.407,A -85,B 0,C 180,E1 -13175.345,E2 -13175.345} C_VEL
LIN {X 0,Y 361.875,Z 539.405,A -85,B 0,C 180,E1 -13179.026,E2 -13179.026} C_VEL
LIN {X 0,Y 361.84,Z 539.375,A -85,B 0,C 180,E1 -13182.829,E2 -13182.829} C_VEL
LIN {X 0,Y 361.863,Z 539.405,A -85,B 0,C 180,E1 -13185.94,E2 -13185.94} C_VEL
LIN {X 0,Y 361.843,Z 539.396,A -85,B 0,C 180,E1 -13189.244,E2 -13189.244} C_VEL
LIN {X 0,Y 361.868,Z 539.407,A -85,B 0,C 180,E1 -13192.777,E2 -13192.777} C_VEL
LIN {X 0,Y 361.859,Z 539.399,A -85,B 0,C 180,E1 -13195.719,E2 -13195.719} C_VEL
LIN {X 0,Y 361.877,Z 539.408,A -85,B 0,C 180,E1 -13199.671,E2 -13199.671} C_VEL
LIN {X 0,Y 361.958,Z 539.396,A -85,B 0,C 180,E1 -13203.475,E2 -13203.475} C_VEL
LIN {X 0,Y 361.988,Z 539.642,A -85,B 0,C 180,E1 -13204.251,E2 -13204.251} C_VEL
LIN {X 0,Y 363.965,Z 549.734,A -85,B 0,C 180,E1 -13207.281,E2 -13207.281} C_VEL
LIN {X 0,Y 364.469,Z 552.251,A -85,B 0,C 180,E1 -13207.942,E2 -13207.942} C_VEL
LIN {X 0,Y 366.565,Z 558.741,A -85,B 0,C 180,E1 -13208.25,E2 -13208.25} C_VEL
LIN {X 0,Y 370.532,Z 578.347,A -85,B 0,C 180,E1 -13208.898,E2 -13208.898} C_VEL
LIN {X 0,Y 369.23,Z 656.96,A -85,B 0,C 180,E1 -13210.434,E2 -13210.434} C_VEL
LIN {X 0,Y 368.817,Z 669.571,A -85,B 0,C 180,E1 -13210.845,E2 -13210.845} C_VEL
LIN {X 0,Y 368.083,Z 682.4,A -85,B 0,C 180,E1 -13211.492,E2 -13211.492} C_VEL
LIN {X 0,Y 367.185,Z 694.251,A -85,B 0,C 180,E1 -13212.31,E2 -13212.31} C_VEL
LIN {X 0,Y 366.221,Z 705.008,A -85,B 0,C 180,E1 -13213.269,E2 -13213.269} C_VEL
LIN {X 0,Y 365.295,Z 715.969,A -85,B 0,C 180,E1 -13214.517,E2 -13214.517} C_VEL
LIN {X 0,Y 364.294,Z 724.869,A -85,B 0,C 180,E1 -13215.76,E2 -13215.76} C_VEL
LIN {X 0,Y 363.287,Z 733.036,A -85,B 0,C 180,E1 -13217.145,E2 -13217.145} C_VEL
LIN {X 0,Y 362.385,Z 741.032,A -85,B 0,C 180,E1 -13218.816,E2 -13218.816} C_VEL
LIN {X 0,Y 361.645,Z 747.452,A -85,B 0,C 180,E1 -13220.491,E2 -13220.491} C_VEL
LIN {X 0,Y 361.118,Z 752.544,A -85,B 0,C 180,E1 -13222.169,E2 -13222.169} C_VEL
LIN {X 0,Y 360.815,Z 756.279,A -85,B 0,C 180,E1 -13223.748,E2 -13223.748} C_VEL
LIN {X 0,Y 360.558,Z 759.408,A -85,B 0,C 180,E1 -13225.527,E2 -13225.527} C_VEL
LIN {X 0,Y 360.418,Z 760.808,A -85,B 0,C 180,E1 -13226.645,E2 -13226.645} C_VEL
LIN {X 0,Y 360.353,Z 762.416,A -85,B 0,C 180,E1 -13228.881,E2 -13228.881} C_VEL
LIN {X 0,Y 360.361,Z 762.649,A -85,B 0,C 180,E1 -13229.999,E2 -13229.999} C_VEL
LIN {X 0,Y 360.353,Z 762.46,A -85,B 0,C 180,E1 -13231.117,E2 -13231.117} C_VEL
LIN {X 0,Y 360.413,Z 760.913,A -85,B 0,C 180,E1 -13233.353,E2 -13233.353} C_VEL
LIN {X 0,Y 360.55,Z 759.557,A -85,B 0,C 180,E1 -13234.471,E2 -13234.471} C_VEL
LIN {X 0,Y 360.793,Z 756.553,A -85,B 0,C 180,E1 -13236.221,E2 -13236.221} C_VEL
LIN {X 0,Y 361.115,Z 752.802,A -85,B 0,C 180,E1 -13237.829,E2 -13237.829} C_VEL
LIN {X 0,Y 361.622,Z 747.79,A -85,B 0,C 180,E1 -13239.507,E2 -13239.507} C_VEL
LIN {X 0,Y 362.311,Z 741.479,A -85,B 0,C 180,E1 -13241.184,E2 -13241.184} C_VEL
LIN {X 0,Y 362.706,Z 738.382,A -85,B 0,C 180,E1 -13241.88,E2 -13241.88} C_VEL
LIN {X 0,Y 362.496,Z 734.883,A -85,B 0,C 180,E1 -13242.632,E2 -13242.632} C_VEL
LIN {X 0,Y 360.47,Z 728.936,A -85,B 0,C 180,E1 -13243.849,E2 -13243.849} C_VEL
LIN {X 0,Y 358.452,Z 722.443,A -85,B 0,C 180,E1 -13245,E2 -13245} C_VEL
LIN {X 0,Y 358.248,Z 718.084,A -85,B 0,C 180,E1 -13245.637,E2 -13245.637} C_VEL
LIN {X 0,Y 359.194,Z 707.619,A -85,B 0,C 180,E1 -13246.905,E2 -13246.905} C_VEL
LIN {X 0,Y 360.379,Z 695.721,A -85,B 0,C 180,E1 -13248.033,E2 -13248.033} C_VEL
LIN {X 0,Y 361.42,Z 683.083,A -85,B 0,C 180,E1 -13248.934,E2 -13248.934} C_VEL
LIN {X 0,Y 362.077,Z 670.444,A -85,B 0,C 180,E1 -13249.598,E2 -13249.598} C_VEL
LIN {X 0,Y 362.631,Z 658.436,A -85,B 0,C 180,E1 -13250.009,E2 -13250.009} C_VEL
LIN {X 0,Y 363.916,Z 578.779,A -85,B 0,C 180,E1 -13251.604,E2 -13251.604} C_VEL
LIN {X 0,Y 359.743,Z 559.151,A -85,B 0,C 180,E1 -13252.285,E2 -13252.285} C_VEL
LIN {X 0,Y 357.355,Z 552.614,A -85,B 0,C 180,E1 -13252.614,E2 -13252.614} C_VEL
LIN {X 0,Y 356.929,Z 550.32,A -85,B 0,C 180,E1 -13253.19,E2 -13253.19} C_VEL
LIN {X 0,Y 354.93,Z 540.352,A -85,B 0,C 180,E1 -13256.297,E2 -13256.297} C_VEL
LIN {X 0,Y 354.816,Z 540.272,A -85,B 0,C 180,E1 -13259.681,E2 -13259.681} C_VEL
LIN {X 0,Y 354.803,Z 540.29,A -85,B 0,C 180,E1 -13263.701,E2 -13263.701} C_VEL
LIN {X 0,Y 354.799,Z 540.284,A -85,B 0,C 180,E1 -13266.458,E2 -13266.458} C_VEL
LIN {X 0,Y 354.82,Z 540.279,A -85,B 0,C 180,E1 -13269.422,E2 -13269.422} C_VEL
LIN {X 0,Y 354.786,Z 540.292,A -85,B 0,C 180,E1 -13272.866,E2 -13272.866} C_VEL
LIN {X 0,Y 354.772,Z 540.287,A -85,B 0,C 180,E1 -13276.104,E2 -13276.104} C_VEL
LIN {X 0,Y 354.82,Z 540.283,A -85,B 0,C 180,E1 -13279.183,E2 -13279.183} C_VEL
LIN {X 0,Y 354.808,Z 540.274,A -85,B 0,C 180,E1 -13282.4,E2 -13282.4} C_VEL
LIN {X 0,Y 354.811,Z 540.287,A -85,B 0,C 180,E1 -13284.94,E2 -13284.94} C_VEL
LIN {X 0,Y 354.788,Z 540.286,A -85,B 0,C 180,E1 -13288.404,E2 -13288.404} C_VEL
LIN {X 0,Y 354.847,Z 540.277,A -85,B 0,C 180,E1 -13291.619,E2 -13291.619} C_VEL
LIN {X 0,Y 354.893,Z 540.276,A -85,B 0,C 180,E1 -13294.172,E2 -13294.172} C_VEL
LIN {X 0,Y 354.828,Z 540.277,A -85,B 0,C 180,E1 -13297.893,E2 -13297.893} C_VEL
LIN {X 0,Y 354.916,Z 540.27,A -85,B 0,C 180,E1 -13301.891,E2 -13301.891} C_VEL
LIN {X 0,Y 354.935,Z 540.271,A -85,B 0,C 180,E1 -13305.981,E2 -13305.981} C_VEL
LIN {X 0,Y 354.97,Z 540.256,A -85,B 0,C 180,E1 -13309.736,E2 -13309.736} C_VEL
LIN {X 0,Y 355.106,Z 540.249,A -85,B 0,C 180,E1 -13312.037,E2 -13312.037} C_VEL
LIN {X 0,Y 355.085,Z 540.251,A -85,B 0,C 180,E1 -13314.321,E2 -13314.321} C_VEL
LIN {X 0,Y 355.238,Z 540.226,A -85,B 0,C 180,E1 -13317.732,E2 -13317.732} C_VEL
LIN {X 0,Y 355.392,Z 540.215,A -85,B 0,C 180,E1 -13320,E2 -13320} C_VEL
LIN {X 0,Y 355.239,Z 540.227,A -85,B 0,C 180,E1 -13322.268,E2 -13322.268} C_VEL
LIN {X 0,Y 355.134,Z 540.245,A -85,B 0,C 180,E1 -13326.819,E2 -13326.819} C_VEL
LIN {X 0,Y 355.008,Z 540.259,A -85,B 0,C 180,E1 -13329.113,E2 -13329.113} C_VEL
LIN {X 0,Y 354.918,Z 540.271,A -85,B 0,C 180,E1 -13332.581,E2 -13332.581} C_VEL
LIN {X 0,Y 354.882,Z 540.269,A -85,B 0,C 180,E1 -13336.096,E2 -13336.096} C_VEL
LIN {X 0,Y 354.901,Z 540.274,A -85,B 0,C 180,E1 -13338.472,E2 -13338.472} C_VEL
LIN {X 0,Y 354.832,Z 540.28,A -85,B 0,C 180,E1 -13342.106,E2 -13342.106} C_VEL
LIN {X 0,Y 354.892,Z 540.272,A -85,B 0,C 180,E1 -13345.828,E2 -13345.828} C_VEL
LIN {X 0,Y 354.811,Z 540.288,A -85,B 0,C 180,E1 -13349.683,E2 -13349.683} C_VEL
LIN {X 0,Y 354.8,Z 540.289,A -85,B 0,C 180,E1 -13353.703,E2 -13353.703} C_VEL
LIN {X 0,Y 354.792,Z 540.268,A -85,B 0,C 180,E1 -13356.46,E2 -13356.46} C_VEL
LIN {X 0,Y 354.818,Z 540.287,A -85,B 0,C 180,E1 -13359.425,E2 -13359.425} C_VEL
LIN {X 0,Y 354.786,Z 540.277,A -85,B 0,C 180,E1 -13362.869,E2 -13362.869} C_VEL
LIN {X 0,Y 354.836,Z 540.279,A -85,B 0,C 180,E1 -13366.116,E2 -13366.116} C_VEL
LIN {X 0,Y 354.852,Z 540.284,A -85,B 0,C 180,E1 -13369.19,E2 -13369.19} C_VEL
LIN {X 0,Y 354.806,Z 540.261,A -85,B 0,C 180,E1 -13372.403,E2 -13372.403} C_VEL
LIN {X 0,Y 354.809,Z 540.29,A -85,B 0,C 180,E1 -13374.942,E2 -13374.942} C_VEL
LIN {X 0,Y 354.786,Z 540.225,A -85,B 0,C 180,E1 -13378.407,E2 -13378.407} C_VEL
LIN {X 0,Y 354.905,Z 540.442,A -85,B 0,C 180,E1 -13379.59,E2 -13379.59} C_VEL
LIN {X 0,Y 357.393,Z 551.806,A -85,B 0,C 180,E1 -13382.738,E2 -13382.738} C_VEL
LIN {X 0,Y 358.906,Z 560.837,A -85,B 0,C 180,E1 -13385.103,E2 -13385.103} C_VEL
LIN {X 0,Y 357.939,Z 570.577,A -85,B 0,C 180,E1 -13387.413,E2 -13387.413} C_VEL
LIN {X 0,Y 358.417,Z 573.83,A -85,B 0,C 180,E1 -13387.578,E2 -13387.578} C_VEL
LIN {X 0,Y 362.722,Z 599.142,A -85,B 0,C 180,E1 -13388.384,E2 -13388.384} C_VEL
LIN {X 0,Y 363.622,Z 604.903,A -85,B 0,C 180,E1 -13388.56,E2 -13388.56} C_VEL
LIN {X 0,Y 362.343,Z 679.032,A -85,B 0,C 180,E1 -13390.048,E2 -13390.048} C_VEL
LIN {X 0,Y 361.589,Z 692.226,A -85,B 0,C 180,E1 -13390.523,E2 -13390.523} C_VEL
LIN {X 0,Y 360.684,Z 705.473,A -85,B 0,C 180,E1 -13391.247,E2 -13391.247} C_VEL
LIN {X 0,Y 359.678,Z 716.606,A -85,B 0,C 180,E1 -13392.078,E2 -13392.078} C_VEL
LIN {X 0,Y 358.504,Z 728.189,A -85,B 0,C 180,E1 -13393.194,E2 -13393.194} C_VEL
LIN {X 0,Y 357.334,Z 739.085,A -85,B 0,C 180,E1 -13394.521,E2 -13394.521} C_VEL
LIN {X 0,Y 356.269,Z 748.832,A -85,B 0,C 180,E1 -13396.017,E2 -13396.017} C_VEL
LIN {X 0,Y 355.153,Z 757.765,A -85,B 0,C 180,E1 -13397.719,E2 -13397.719} C_VEL
LIN {X 0,Y 354.392,Z 764.959,A -85,B 0,C 180,E1 -13399.431,E2 -13399.431} C_VEL
LIN {X 0,Y 353.9,Z 769.814,A -85,B 0,C 180,E1 -13400.86,E2 -13400.86} C_VEL
LIN {X 0,Y 353.519,Z 774.536,A -85,B 0,C 180,E1 -13402.577,E2 -13402.577} C_VEL
LIN {X 0,Y 353.281,Z 778.149,A -85,B 0,C 180,E1 -13404.293,E2 -13404.293} C_VEL
LIN {X 0,Y 353.28,Z 780.014,A -85,B 0,C 180,E1 -13405.437,E2 -13405.437} C_VEL
LIN {X 0,Y 353.223,Z 781.409,A -85,B 0,C 180,E1 -13406.579,E2 -13406.579} C_VEL
LIN {X 0,Y 353.222,Z 784.384,A -85,B 0,C 180,E1 -13410.001,E2 -13410.001} C_VEL
LIN {X 0,Y 353.167,Z 784.67,A -85,B 0,C 180,E1 -13411.141,E2 -13411.141} C_VEL
LIN {X 0,Y 353.169,Z 784.33,A -85,B 0,C 180,E1 -13412.282,E2 -13412.282} C_VEL
LIN {X 0,Y 353.227,Z 783.371,A -85,B 0,C 180,E1 -13413.423,E2 -13413.423} C_VEL
LIN {X 0,Y 353.326,Z 780.837,A -85,B 0,C 180,E1 -13415.136,E2 -13415.136} C_VEL
LIN {X 0,Y 353.4,Z 778.346,A -85,B 0,C 180,E1 -13416.28,E2 -13416.28} C_VEL
LIN {X 0,Y 353.902,Z 769.773,A -85,B 0,C 180,E1 -13419.142,E2 -13419.142} C_VEL
LIN {X 0,Y 354.594,Z 762.666,A -85,B 0,C 180,E1 -13421.143,E2 -13421.143} C_VEL
LIN {X 0,Y 355.509,Z 754.959,A -85,B 0,C 180,E1 -13422.851,E2 -13422.851} C_VEL
LIN {X 0,Y 356.598,Z 745.28,A -85,B 0,C 180,E1 -13424.554,E2 -13424.554} C_VEL
LIN {X 0,Y 357.676,Z 735.298,A -85,B 0,C 180,E1 -13425.968,E2 -13425.968} C_VEL
LIN {X 0,Y 358.888,Z 724.021,A -85,B 0,C 180,E1 -13427.23,E2 -13427.23} C_VEL
LIN {X 0,Y 360.01,Z 712.981,A -85,B 0,C 180,E1 -13428.202,E2 -13428.202} C_VEL
LIN {X 0,Y 361.008,Z 700.744,A -85,B 0,C 180,E1 -13429.032,E2 -13429.032} C_VEL
LIN {X 0,Y 361.876,Z 687.86,A -85,B 0,C 180,E1 -13429.648,E2 -13429.648} C_VEL
LIN {X 0,Y 362.411,Z 674.149,A -85,B 0,C 180,E1 -13430.061,E2 -13430.061} C_VEL
LIN {X 0,Y 363.561,Z 604.806,A -85,B 0,C 180,E1 -13431.433,E2 -13431.433} C_VEL
LIN {X 0,Y 359.035,Z 576.978,A -85,B 0,C 180,E1 -13432.31,E2 -13432.31} C_VEL
LIN {X 0,Y 358.801,Z 572.595,A -85,B 0,C 180,E1 -13432.74,E2 -13432.74} C_VEL
LIN {X 0,Y 358.356,Z 567.25,A -85,B 0,C 180,E1 -13433.4,E2 -13433.4} C_VEL
LIN {X 0,Y 358.897,Z 560.76,A -85,B 0,C 180,E1 -13434.9,E2 -13434.9} C_VEL
LIN {X 0,Y 357.091,Z 550.237,A -85,B 0,C 180,E1 -13437.667,E2 -13437.667} C_VEL
LIN {X 0,Y 354.866,Z 540.353,A -85,B 0,C 180,E1 -13440.457,E2 -13440.457} C_VEL
LIN {X 0,Y 354.81,Z 540.287,A -85,B 0,C 180,E1 -13443.703,E2 -13443.703} C_VEL
LIN {X 0,Y 354.802,Z 540.29,A -85,B 0,C 180,E1 -13446.46,E2 -13446.46} C_VEL
LIN {X 0,Y 354.828,Z 540.285,A -85,B 0,C 180,E1 -13449.424,E2 -13449.424} C_VEL
LIN {X 0,Y 354.792,Z 540.289,A -85,B 0,C 180,E1 -13452.868,E2 -13452.868} C_VEL
LIN {X 0,Y 354.771,Z 540.292,A -85,B 0,C 180,E1 -13456.104,E2 -13456.104} C_VEL
LIN {X 0,Y 354.792,Z 540.29,A -85,B 0,C 180,E1 -13459.179,E2 -13459.179} C_VEL
LIN {X 0,Y 354.864,Z 540.519,A -85,B 0,C 180,E1 -13462.504,E2 -13462.504} C_VEL
LIN {X 0,Y 356.503,Z 544.573,A -85,B 0,C 180,E1 -13463.928,E2 -13463.928} C_VEL
LIN {X 0,Y 359.494,Z 552.585,A -85,B 0,C 180,E1 -13466.376,E2 -13466.376} C_VEL
LIN {X 0,Y 362.092,Z 561.113,A -85,B 0,C 180,E1 -13468.652,E2 -13468.652} C_VEL
LIN {X 0,Y 363.862,Z 569.288,A -85,B 0,C 180,E1 -13470.588,E2 -13470.588} C_VEL
LIN {X 0,Y 364.128,Z 573.473,A -85,B 0,C 180,E1 -13471.465,E2 -13471.465} C_VEL
